LIN {X -0.120,Y -569.299,Z 835.308,A 0.000,B 0.000,C 90.000,E1 91.489} C_DIS
LIN {X -0.052,Y -569.722,Z 835.301,A 0.000,B 0.000,C 90.000,E1 90.115} C_DIS
LIN {X 0.024,Y -570.053,Z 835.293,A 0.000,B 0.000,C 90.000,E1 88.740} C_DIS
LIN {X -0.168,Y -570.463,Z 835.282,A 0.000,B 0.000,C 90.000,E1 86.846} C_DIS
LIN {X 0.104,Y -570.739,Z 835.273,A 0.000,B 0.000,C 90.000,E1 85.179} C_DIS
LIN {X -0.200,Y -571.053,Z 835.264,A 0.000,B 0.000,C 90.000,E1 83.571} C_DIS
LIN {X 0.004,Y -571.342,Z 835.257,A 0.000,B 0.000,C 90.000,E1 82.186} C_DIS
LIN {X -0.074,Y -571.786,Z 835.248,A 0.000,B 0.000,C 90.000,E1 80.557} C_DIS
LIN {X 0.064,Y -572.418,Z 835.237,A 0.000,B 0.000,C 90.000,E1 78.634} C_DIS
LIN {X -0.068,Y -572.823,Z 835.229,A 0.000,B 0.000,C 90.000,E1 77.285} C_DIS
LIN {X -0.005,Y -573.147,Z 835.220,A 0.000,B 0.000,C 90.000,E1 75.644} C_DIS
LIN {X -0.194,Y -573.354,Z 835.214,A 0.000,B 0.000,C 90.000,E1 74.574} C_DIS
LIN {X -0.035,Y -573.431,Z 835.204,A 0.000,B 0.000,C 90.000,E1 72.653} C_DIS
LIN {X 0.133,Y -573.360,Z 835.196,A 0.000,B 0.000,C 90.000,E1 71.275} C_DIS
LIN {X 0.102,Y -573.177,Z 835.187,A 0.000,B 0.000,C 90.000,E1 69.645} C_DIS
LIN {X -0.261,Y -573.034,Z 835.181,A 0.000,B 0.000,C 90.000,E1 68.592} C_DIS
LIN {X -0.090,Y -572.851,Z 835.175,A 0.000,B 0.000,C 90.000,E1 67.486} C_DIS
LIN {X 0.133,Y -572.485,Z 835.167,A 0.000,B 0.000,C 90.000,E1 66.102} C_DIS
LIN {X 0.191,Y -571.841,Z 835.158,A 0.000,B 0.000,C 90.000,E1 64.460} C_DIS
LIN {X -0.118,Y -571.242,Z 835.151,A 0.000,B 0.000,C 90.000,E1 63.127} C_DIS
LIN {X -0.183,Y -570.569,Z 835.143,A 0.000,B 0.000,C 90.000,E1 61.769} C_DIS
LIN {X 0.251,Y -570.332,Z 835.140,A 0.000,B 0.000,C 90.000,E1 61.179} C_DIS
LIN {X -0.159,Y -569.417,Z 835.134,A 0.000,B 0.000,C 90.000,E1 60.127} C_DIS
LIN {X 0.013,Y -568.014,Z 835.126,A 0.000,B 0.000,C 90.000,E1 58.742} C_DIS
LIN {X -0.031,Y -566.388,Z 835.119,A 0.000,B 0.000,C 90.000,E1 57.375} C_DIS
LIN {X -0.208,Y -564.795,Z 835.113,A 0.000,B 0.000,C 90.000,E1 56.294} C_DIS
LIN {X -0.203,Y -563.469,Z 835.108,A 0.000,B 0.000,C 90.000,E1 55.468} C_DIS
LIN {X -0.115,Y -561.414,Z 835.102,A 0.000,B 0.000,C 90.000,E1 54.356} C_DIS
LIN {X 0.176,Y -559.714,Z 835.097,A 0.000,B 0.000,C 90.000,E1 53.497} C_DIS
LIN {X -0.086,Y -558.502,Z 835.094,A 0.000,B 0.000,C 90.000,E1 52.970} C_DIS
LIN {X 0.179,Y -556.410,Z 835.090,A 0.000,B 0.000,C 90.000,E1 52.110} C_DIS
LIN {X -0.019,Y -554.074,Z 835.085,A 0.000,B 0.000,C 90.000,E1 51.295} C_DIS
LIN {X 0.124,Y -552.393,Z 835.082,A 0.000,B 0.000,C 90.000,E1 50.723} C_DIS
LIN {X -0.116,Y -549.571,Z 835.077,A 0.000,B 0.000,C 90.000,E1 49.908} C_DIS
LIN {X -0.027,Y -546.387,Z 835.073,A 0.000,B 0.000,C 90.000,E1 49.057} C_DIS
LIN {X 0.242,Y -543.489,Z 835.069,A 0.000,B 0.000,C 90.000,E1 48.324} C_DIS
LIN {X -0.118,Y -540.968,Z 835.065,A 0.000,B 0.000,C 90.000,E1 47.796} C_DIS
LIN {X -0.130,Y -538.213,Z 835.062,A 0.000,B 0.000,C 90.000,E1 47.229} C_DIS
LIN {X 0.020,Y -534.370,Z 835.058,A 0.000,B 0.000,C 90.000,E1 46.500} C_DIS
LIN {X 0.349,Y -531.058,Z 835.055,A 0.000,B 0.000,C 90.000,E1 45.891} C_DIS
LIN {X 0.268,Y -527.360,Z 835.052,A 0.000,B 0.000,C 90.000,E1 45.324} C_DIS
LIN {X 0.161,Y -523.332,Z 835.049,A 0.000,B 0.000,C 90.000,E1 44.757} C_DIS
LIN {X 0.026,Y -518.943,Z 835.046,A 0.000,B 0.000,C 90.000,E1 44.190} C_DIS
LIN {X -0.024,Y -514.327,Z 835.042,A 0.000,B 0.000,C 90.000,E1 43.623} C_DIS
LIN {X 0.089,Y -510.741,Z 835.040,A 0.000,B 0.000,C 90.000,E1 43.176} C_DIS
LIN {X 0.028,Y -505.522,Z 835.037,A 0.000,B 0.000,C 90.000,E1 42.609} C_DIS
LIN {X -0.024,Y -500.041,Z 835.034,A 0.000,B 0.000,C 90.000,E1 42.043} C_DIS
LIN {X 0.016,Y -496.033,Z 835.031,A 0.000,B 0.000,C 90.000,E1 41.634} C_DIS
LIN {X 0.029,Y -489.092,Z 835.028,A 0.000,B 0.000,C 90.000,E1 40.987} C_DIS
LIN {X 0.092,Y -483.021,Z 835.025,A 0.000,B 0.000,C 90.000,E1 40.458} C_DIS
LIN {X -0.032,Y -475.383,Z 835.021,A 0.000,B 0.000,C 90.000,E1 39.850} C_DIS
LIN {X 0.137,Y -466.165,Z 835.017,A 0.000,B 0.000,C 90.000,E1 39.116} C_DIS
LIN {X 0.072,Y -453.584,Z 835.012,A 0.000,B 0.000,C 90.000,E1 38.177} C_DIS
LIN {X 0.015,Y -440.852,Z 835.007,A 0.000,B 0.000,C 90.000,E1 37.237} C_DIS
LIN {X 0.060,Y -420.752,Z 834.998,A 0.000,B 0.000,C 90.000,E1 35.644} C_DIS
LIN {X 0.124,Y -410.398,Z 834.993,A 0.000,B 0.000,C 90.000,E1 34.739} C_DIS
LIN {X -0.033,Y -404.337,Z 834.990,A 0.000,B 0.000,C 90.000,E1 34.199} C_DIS
LIN {X 0.112,Y -399.570,Z 834.987,A 0.000,B 0.000,C 90.000,E1 33.658} C_DIS
LIN {X 0.091,Y -398.266,Z 834.986,A 0.000,B 0.000,C 90.000,E1 33.499} C_DIS
LIN {X -0.239,Y -395.679,Z 834.984,A 0.000,B 0.000,C 90.000,E1 33.166} C_DIS
LIN {X 0.055,Y -395.661,Z 834.984,A 0.000,B 0.000,C 90.000,E1 33.118} C_DIS
LIN {X 0.091,Y -393.941,Z 834.977,A 0.000,B 0.000,C 90.000,E1 31.926} C_DIS
LIN {X -0.123,Y -391.263,Z 834.970,A 0.000,B 0.000,C 90.000,E1 30.541} C_DIS
LIN {X -0.028,Y -391.514,Z 834.964,A 0.000,B 0.000,C 90.000,E1 29.461} C_DIS
LIN {X -0.208,Y -392.887,Z 834.950,A 0.000,B 0.000,C 90.000,E1 27.001} C_DIS
LIN {X 0.035,Y -394.828,Z 834.934,A 0.000,B 0.000,C 90.000,E1 24.131} C_DIS
LIN {X -0.055,Y -396.510,Z 834.922,A 0.000,B 0.000,C 90.000,E1 22.025} C_DIS
LIN {X -0.016,Y -399.373,Z 834.905,A 0.000,B 0.000,C 90.000,E1 18.852} C_DIS
LIN {X -0.132,Y -402.980,Z 834.887,A 0.000,B 0.000,C 90.000,E1 15.717} C_DIS
LIN {X -0.166,Y -407.456,Z 834.870,A 0.000,B 0.000,C 90.000,E1 12.591} C_DIS
LIN {X 0.029,Y -410.786,Z 834.858,A 0.000,B 0.000,C 90.000,E1 10.489} C_DIS
LIN {X -0.210,Y -413.708,Z 834.849,A 0.000,B 0.000,C 90.000,E1 8.803} C_DIS
LIN {X 0.007,Y -417.352,Z 834.837,A 0.000,B 0.000,C 90.000,E1 6.720} C_DIS
LIN {X -0.070,Y -422.343,Z 834.822,A 0.000,B 0.000,C 90.000,E1 4.012} C_DIS
LIN {X 0.044,Y -429.232,Z 834.804,A 0.000,B 0.000,C 90.000,E1 0.630} C_DIS
LIN {X -0.189,Y -435.722,Z 834.788,A 0.000,B 0.000,C 90.000,E1 357.822} C_DIS
LIN {X 0.132,Y -441.316,Z 834.775,A 0.000,B 0.000,C 90.000,E1 355.469} C_DIS
LIN {X 0.065,Y -446.342,Z 834.764,A 0.000,B 0.000,C 90.000,E1 353.514} C_DIS
LIN {X 0.097,Y -449.017,Z 834.759,A 0.000,B 0.000,C 90.000,E1 352.534} C_DIS
LIN {X -0.037,Y -450.535,Z 834.756,A 0.000,B 0.000,C 90.000,E1 352.064} C_DIS
LIN {X -0.192,Y -453.090,Z 834.753,A 0.000,B 0.000,C 90.000,E1 351.489} C_DIS
LIN {X -0.176,Y -455.431,Z 834.750,A 0.000,B 0.000,C 90.000,E1 351.084} C_DIS
LIN {X -0.065,Y -460.510,Z 834.748,A 0.000,B 0.000,C 90.000,E1 350.557} C_DIS
LIN {X -0.105,Y -466.031,Z 834.745,A 0.000,B 0.000,C 90.000,E1 350.151} C_DIS
LIN {X 0.110,Y -480.162,Z 834.741,A 0.000,B 0.000,C 90.000,E1 349.285} C_DIS
LIN {X 0.120,Y -489.899,Z 834.737,A 0.000,B 0.000,C 90.000,E1 348.701} C_DIS
LIN {X 0.257,Y -496.316,Z 834.735,A 0.000,B 0.000,C 90.000,E1 348.285} C_DIS
LIN {X -0.026,Y -507.454,Z 834.731,A 0.000,B 0.000,C 90.000,E1 347.589} C_DIS
LIN {X 0.093,Y -516.832,Z 834.728,A 0.000,B 0.000,C 90.000,E1 346.937} C_DIS
LIN {X 0.112,Y -527.555,Z 834.723,A 0.000,B 0.000,C 90.000,E1 346.172} C_DIS
LIN {X -0.180,Y -535.027,Z 834.720,A 0.000,B 0.000,C 90.000,E1 345.644} C_DIS
LIN {X 0.184,Y -542.141,Z 834.717,A 0.000,B 0.000,C 90.000,E1 345.046} C_DIS
LIN {X 0.110,Y -549.312,Z 834.714,A 0.000,B 0.000,C 90.000,E1 344.464} C_DIS
LIN {X -0.045,Y -558.907,Z 834.709,A 0.000,B 0.000,C 90.000,E1 343.614} C_DIS
LIN {X -0.022,Y -565.482,Z 834.705,A 0.000,B 0.000,C 90.000,E1 342.960} C_DIS
LIN {X -0.185,Y -571.704,Z 834.702,A 0.000,B 0.000,C 90.000,E1 342.308} C_DIS
LIN {X 0.160,Y -578.789,Z 834.697,A 0.000,B 0.000,C 90.000,E1 341.456} C_DIS
LIN {X 0.191,Y -583.083,Z 834.694,A 0.000,B 0.000,C 90.000,E1 340.913} C_DIS
LIN {X -0.150,Y -590.010,Z 834.689,A 0.000,B 0.000,C 90.000,E1 340.007} C_DIS
LIN {X -0.159,Y -595.400,Z 834.684,A 0.000,B 0.000,C 90.000,E1 339.209} C_DIS
LIN {X -0.110,Y -600.400,Z 834.680,A 0.000,B 0.000,C 90.000,E1 338.411} C_DIS
LIN {X 0.288,Y -603.548,Z 834.677,A 0.000,B 0.000,C 90.000,E1 337.847} C_DIS
LIN {X 0.345,Y -610.264,Z 834.671,A 0.000,B 0.000,C 90.000,E1 336.666} C_DIS
LIN {X -0.032,Y -615.315,Z 834.666,A 0.000,B 0.000,C 90.000,E1 335.793} C_DIS
LIN {X -0.098,Y -620.112,Z 834.661,A 0.000,B 0.000,C 90.000,E1 334.897} C_DIS
LIN {X 0.184,Y -623.975,Z 834.656,A 0.000,B 0.000,C 90.000,E1 334.101} C_DIS
LIN {X 0.211,Y -627.690,Z 834.652,A 0.000,B 0.000,C 90.000,E1 333.332} C_DIS
LIN {X -0.262,Y -632.292,Z 834.646,A 0.000,B 0.000,C 90.000,E1 332.359} C_DIS
LIN {X 0.230,Y -637.757,Z 834.639,A 0.000,B 0.000,C 90.000,E1 331.051} C_DIS
LIN {X -0.174,Y -640.869,Z 834.635,A 0.000,B 0.000,C 90.000,E1 330.333} C_DIS
LIN {X -0.096,Y -645.795,Z 834.628,A 0.000,B 0.000,C 90.000,E1 329.076} C_DIS
LIN {X -0.020,Y -649.321,Z 834.623,A 0.000,B 0.000,C 90.000,E1 328.074} C_DIS
LIN {X -0.014,Y -653.497,Z 834.616,A 0.000,B 0.000,C 90.000,E1 326.834} C_DIS
LIN {X 0.062,Y -655.742,Z 834.612,A 0.000,B 0.000,C 90.000,E1 326.087} C_DIS
LIN {X 0.083,Y -658.634,Z 834.606,A 0.000,B 0.000,C 90.000,E1 325.102} C_DIS
LIN {X 0.145,Y -661.300,Z 834.601,A 0.000,B 0.000,C 90.000,E1 324.116} C_DIS
LIN {X -0.251,Y -663.053,Z 834.597,A 0.000,B 0.000,C 90.000,E1 323.417} C_DIS
LIN {X 0.263,Y -665.237,Z 834.591,A 0.000,B 0.000,C 90.000,E1 322.396} C_DIS
LIN {X -0.125,Y -667.211,Z 834.586,A 0.000,B 0.000,C 90.000,E1 321.457} C_DIS
LIN {X -0.069,Y -668.989,Z 834.580,A 0.000,B 0.000,C 90.000,E1 320.481} C_DIS
LIN {X 0.090,Y -670.998,Z 834.574,A 0.000,B 0.000,C 90.000,E1 319.256} C_DIS
LIN {X 0.230,Y -673.653,Z 834.564,A 0.000,B 0.000,C 90.000,E1 317.553} C_DIS
LIN {X -0.165,Y -674.737,Z 834.560,A 0.000,B 0.000,C 90.000,E1 316.863} C_DIS
LIN {X 0.035,Y -676.870,Z 834.551,A 0.000,B 0.000,C 90.000,E1 315.162} C_DIS
LIN {X 0.212,Y -678.249,Z 834.544,A 0.000,B 0.000,C 90.000,E1 313.947} C_DIS
LIN {X -0.020,Y -679.817,Z 834.536,A 0.000,B 0.000,C 90.000,E1 312.528} C_DIS
LIN {X 0.279,Y -681.355,Z 834.528,A 0.000,B 0.000,C 90.000,E1 311.067} C_DIS
LIN {X 0.119,Y -682.528,Z 834.522,A 0.000,B 0.000,C 90.000,E1 309.886} C_DIS
LIN {X -0.014,Y -683.593,Z 834.515,A 0.000,B 0.000,C 90.000,E1 308.705} C_DIS
LIN {X -0.135,Y -684.639,Z 834.508,A 0.000,B 0.000,C 90.000,E1 307.523} C_DIS
LIN {X 0.297,Y -685.662,Z 834.502,A 0.000,B 0.000,C 90.000,E1 306.297} C_DIS
LIN {X 0.340,Y -686.618,Z 834.495,A 0.000,B 0.000,C 90.000,E1 305.105} C_DIS
LIN {X 0.027,Y -687.625,Z 834.487,A 0.000,B 0.000,C 90.000,E1 303.706} C_DIS
LIN {X -0.073,Y -688.603,Z 834.479,A 0.000,B 0.000,C 90.000,E1 302.291} C_DIS
LIN {X 0.433,Y -689.807,Z 834.470,A 0.000,B 0.000,C 90.000,E1 300.590} C_DIS
LIN {X 0.021,Y -690.884,Z 834.462,A 0.000,B 0.000,C 90.000,E1 299.205} C_DIS
LIN {X -0.006,Y -691.825,Z 834.456,A 0.000,B 0.000,C 90.000,E1 298.025} C_DIS
LIN {X -0.227,Y -693.391,Z 834.445,A 0.000,B 0.000,C 90.000,E1 296.155} C_DIS
LIN {X 0.292,Y -694.802,Z 834.436,A 0.000,B 0.000,C 90.000,E1 294.463} C_DIS
LIN {X 0.126,Y -695.027,Z 834.432,A 0.000,B 0.000,C 90.000,E1 293.770} C_DIS
LIN {X -0.290,Y -694.417,Z 834.430,A 0.000,B 0.000,C 90.000,E1 293.334} C_DIS
LIN {X -0.042,Y -693.967,Z 834.428,A 0.000,B 0.000,C 90.000,E1 293.078} C_DIS
LIN {X 0.056,Y -692.154,Z 834.426,A 0.000,B 0.000,C 90.000,E1 292.717} C_DIS
LIN {X 0.295,Y -690.711,Z 834.425,A 0.000,B 0.000,C 90.000,E1 292.461} C_DIS
LIN {X -0.226,Y -689.876,Z 834.424,A 0.000,B 0.000,C 90.000,E1 292.386} C_DIS
LIN {X -0.111,Y -688.662,Z 834.424,A 0.000,B 0.000,C 90.000,E1 292.259} C_DIS
LIN {X -0.186,Y -684.038,Z 834.422,A 0.000,B 0.000,C 90.000,E1 291.950} C_DIS
LIN {X -0.073,Y -682.425,Z 834.421,A 0.000,B 0.000,C 90.000,E1 291.844} C_DIS
LIN {X 0.292,Y -680.489,Z 834.421,A 0.000,B 0.000,C 90.000,E1 291.716} C_DIS
LIN {X 0.211,Y -671.837,Z 834.419,A 0.000,B 0.000,C 90.000,E1 291.461} C_DIS
LIN {X 0.243,Y -663.448,Z 834.418,A 0.000,B 0.000,C 90.000,E1 291.280} C_DIS
LIN {X 0.212,Y -655.251,Z 834.418,A 0.000,B 0.000,C 90.000,E1 291.153} C_DIS
LIN {X 0.175,Y -646.300,Z 834.417,A 0.000,B 0.000,C 90.000,E1 290.972} C_DIS
LIN {X 0.364,Y -639.749,Z 834.416,A 0.000,B 0.000,C 90.000,E1 290.791} C_DIS
LIN {X 0.255,Y -635.161,Z 834.415,A 0.000,B 0.000,C 90.000,E1 290.663} C_DIS
LIN {X -0.113,Y -631.474,Z 834.414,A 0.000,B 0.000,C 90.000,E1 290.556} C_DIS
LIN {X -0.036,Y -626.194,Z 834.413,A 0.000,B 0.000,C 90.000,E1 290.301} C_DIS
LIN {X -0.165,Y -625.101,Z 834.412,A 0.000,B 0.000,C 90.000,E1 290.248} C_DIS
LIN {X 0.250,Y -623.492,Z 834.412,A 0.000,B 0.000,C 90.000,E1 290.066} C_DIS
LIN {X 0.217,Y -623.471,Z 834.412,A 0.000,B 0.000,C 90.000,E1 290.066} C_DIS
LIN {X 0.049,Y -623.220,Z 834.411,A 0.000,B 0.000,C 90.000,E1 289.939} C_DIS
LIN {X -0.061,Y -623.280,Z 834.411,A 0.000,B 0.000,C 90.000,E1 289.885} C_DIS
LIN {X -0.190,Y -624.798,Z 834.408,A 0.000,B 0.000,C 90.000,E1 289.450} C_DIS
LIN {X -0.067,Y -629.481,Z 834.403,A 0.000,B 0.000,C 90.000,E1 288.598} C_DIS
LIN {X -0.155,Y -632.392,Z 834.401,A 0.000,B 0.000,C 90.000,E1 288.109} C_DIS
LIN {X 0.128,Y -636.087,Z 834.396,A 0.000,B 0.000,C 90.000,E1 287.330} C_DIS
LIN {X -0.232,Y -638.364,Z 834.394,A 0.000,B 0.000,C 90.000,E1 286.858} C_DIS
LIN {X 0.055,Y -641.172,Z 834.389,A 0.000,B 0.000,C 90.000,E1 286.079} C_DIS
LIN {X 0.197,Y -643.583,Z 834.385,A 0.000,B 0.000,C 90.000,E1 285.315} C_DIS
LIN {X 0.061,Y -644.904,Z 834.382,A 0.000,B 0.000,C 90.000,E1 284.828} C_DIS
LIN {X 0.246,Y -646.463,Z 834.378,A 0.000,B 0.000,C 90.000,E1 284.064} C_DIS
LIN {X -0.039,Y -647.380,Z 834.376,A 0.000,B 0.000,C 90.000,E1 283.592} C_DIS
LIN {X 0.313,Y -647.948,Z 834.373,A 0.000,B 0.000,C 90.000,E1 283.063} C_DIS
LIN {X -0.100,Y -648.147,Z 834.369,A 0.000,B 0.000,C 90.000,E1 282.355} C_DIS
LIN {X 0.256,Y -648.026,Z 834.366,A 0.000,B 0.000,C 90.000,E1 281.827} C_DIS
LIN {X -0.151,Y -647.731,Z 834.363,A 0.000,B 0.000,C 90.000,E1 281.366} C_DIS
LIN {X 0.061,Y -646.822,Z 834.359,A 0.000,B 0.000,C 90.000,E1 280.602} C_DIS
LIN {X -0.344,Y -645.875,Z 834.356,A 0.000,B 0.000,C 90.000,E1 280.141} C_DIS
LIN {X -0.005,Y -644.634,Z 834.353,A 0.000,B 0.000,C 90.000,E1 279.613} C_DIS
LIN {X 0.217,Y -642.910,Z 834.351,A 0.000,B 0.000,C 90.000,E1 279.095} C_DIS
LIN {X -0.107,Y -640.802,Z 834.348,A 0.000,B 0.000,C 90.000,E1 278.624} C_DIS
LIN {X 0.094,Y -638.380,Z 834.345,A 0.000,B 0.000,C 90.000,E1 278.106} C_DIS
LIN {X -0.221,Y -636.307,Z 834.343,A 0.000,B 0.000,C 90.000,E1 277.757} C_DIS
LIN {X 0.085,Y -633.884,Z 834.341,A 0.000,B 0.000,C 90.000,E1 277.352} C_DIS
LIN {X 0.093,Y -629.125,Z 834.337,A 0.000,B 0.000,C 90.000,E1 276.720} C_DIS
LIN {X -0.263,Y -625.775,Z 834.335,A 0.000,B 0.000,C 90.000,E1 276.372} C_DIS
LIN {X 0.212,Y -624.546,Z 834.335,A 0.000,B 0.000,C 90.000,E1 276.201} C_DIS
LIN {X 0.028,Y -619.077,Z 834.332,A 0.000,B 0.000,C 90.000,E1 275.739} C_DIS
LIN {X 0.263,Y -613.057,Z 834.330,A 0.000,B 0.000,C 90.000,E1 275.277} C_DIS
LIN {X -0.060,Y -609.758,Z 834.328,A 0.000,B 0.000,C 90.000,E1 275.106} C_DIS
LIN {X 0.103,Y -604.710,Z 834.327,A 0.000,B 0.000,C 90.000,E1 274.821} C_DIS
LIN {X -0.280,Y -597.826,Z 834.325,A 0.000,B 0.000,C 90.000,E1 274.531} C_DIS
LIN {X 0.231,Y -590.869,Z 834.323,A 0.000,B 0.000,C 90.000,E1 274.188} C_DIS
LIN {X -0.065,Y -585.648,Z 834.322,A 0.000,B 0.000,C 90.000,E1 274.012} C_DIS
LIN {X -0.120,Y -579.728,Z 834.321,A 0.000,B 0.000,C 90.000,E1 273.841} C_DIS
LIN {X -0.062,Y -577.758,Z 834.321,A 0.000,B 0.000,C 90.000,E1 273.784} C_DIS
LIN {X -0.149,Y -571.161,Z 834.320,A 0.000,B 0.000,C 90.000,E1 273.669} C_DIS
LIN {X -0.186,Y -564.612,Z 834.320,A 0.000,B 0.000,C 90.000,E1 273.612} C_DIS
LIN {X 0.085,Y -553.744,Z 834.320,A 0.000,B 0.000,C 90.000,E1 273.555} C_DIS
LIN {X -0.236,Y -552.354,Z 834.320,A 0.000,B 0.000,C 90.000,E1 273.555} C_DIS
LIN {X 0.260,Y -550.562,Z 834.319,A 0.000,B 0.000,C 90.000,E1 273.440} C_DIS
LIN {X 0.217,Y -550.542,Z 834.319,A 0.000,B 0.000,C 90.000,E1 273.440} C_DIS
LIN {X -0.216,Y -549.459,Z 834.318,A 0.000,B 0.000,C 90.000,E1 273.212} C_DIS
LIN {X 0.099,Y -548.692,Z 834.316,A 0.000,B 0.000,C 90.000,E1 272.808} C_DIS
LIN {X -0.191,Y -547.087,Z 834.308,A 0.000,B 0.000,C 90.000,E1 271.432} C_DIS
LIN {X 0.191,Y -545.161,Z 834.294,A 0.000,B 0.000,C 90.000,E1 268.854} C_DIS
LIN {X -0.123,Y -543.975,Z 834.284,A 0.000,B 0.000,C 90.000,E1 267.192} C_DIS
LIN {X 0.086,Y -543.031,Z 834.276,A 0.000,B 0.000,C 90.000,E1 265.755} C_DIS
LIN {X -0.245,Y -541.924,Z 834.267,A 0.000,B 0.000,C 90.000,E1 264.090} C_DIS
LIN {X -0.097,Y -541.269,Z 834.262,A 0.000,B 0.000,C 90.000,E1 263.223} C_DIS
LIN {X 0.113,Y -539.960,Z 834.254,A 0.000,B 0.000,C 90.000,E1 261.781} C_DIS
LIN {X -0.089,Y -538.416,Z 834.245,A 0.000,B 0.000,C 90.000,E1 260.095} C_DIS
LIN {X 0.306,Y -536.679,Z 834.235,A 0.000,B 0.000,C 90.000,E1 258.342} C_DIS
LIN {X 0.135,Y -534.959,Z 834.226,A 0.000,B 0.000,C 90.000,E1 256.645} C_DIS
LIN {X -0.051,Y -533.642,Z 834.220,A 0.000,B 0.000,C 90.000,E1 255.519} C_DIS
LIN {X -0.216,Y -532.003,Z 834.212,A 0.000,B 0.000,C 90.000,E1 254.102} C_DIS
LIN {X -0.115,Y -530.321,Z 834.204,A 0.000,B 0.000,C 90.000,E1 252.653} C_DIS
LIN {X 0.287,Y -528.962,Z 834.197,A 0.000,B 0.000,C 90.000,E1 251.456} C_DIS
LIN {X 0.157,Y -527.447,Z 834.191,A 0.000,B 0.000,C 90.000,E1 250.315} C_DIS
LIN {X -0.144,Y -525.445,Z 834.183,A 0.000,B 0.000,C 90.000,E1 248.901} C_DIS
LIN {X 0.051,Y -522.569,Z 834.171,A 0.000,B 0.000,C 90.000,E1 246.847} C_DIS
LIN {X -0.127,Y -520.299,Z 834.163,A 0.000,B 0.000,C 90.000,E1 245.409} C_DIS
LIN {X -0.026,Y -518.493,Z 834.157,A 0.000,B 0.000,C 90.000,E1 244.229} C_DIS
LIN {X 0.033,Y -516.490,Z 834.150,A 0.000,B 0.000,C 90.000,E1 243.050} C_DIS
LIN {X -0.154,Y -513.368,Z 834.141,A 0.000,B 0.000,C 90.000,E1 241.307} C_DIS
LIN {X 0.187,Y -510.651,Z 834.132,A 0.000,B 0.000,C 90.000,E1 239.793} C_DIS
LIN {X 0.135,Y -508.458,Z 834.126,A 0.000,B 0.000,C 90.000,E1 238.614} C_DIS
LIN {X -0.119,Y -506.168,Z 834.119,A 0.000,B 0.000,C 90.000,E1 237.454} C_DIS
LIN {X -0.096,Y -503.039,Z 834.111,A 0.000,B 0.000,C 90.000,E1 235.960} C_DIS
LIN {X -0.147,Y -500.340,Z 834.104,A 0.000,B 0.000,C 90.000,E1 234.769} C_DIS
LIN {X 0.194,Y -496.097,Z 834.094,A 0.000,B 0.000,C 90.000,E1 232.924} C_DIS
LIN {X -0.055,Y -493.286,Z 834.087,A 0.000,B 0.000,C 90.000,E1 231.743} C_DIS
LIN {X 0.026,Y -487.613,Z 834.074,A 0.000,B 0.000,C 90.000,E1 229.299} C_DIS
LIN {X -0.026,Y -484.748,Z 834.067,A 0.000,B 0.000,C 90.000,E1 228.081} C_DIS
LIN {X 0.261,Y -479.909,Z 834.055,A 0.000,B 0.000,C 90.000,E1 225.891} C_DIS
LIN {X 0.295,Y -475.883,Z 834.045,A 0.000,B 0.000,C 90.000,E1 224.028} C_DIS
LIN {X 0.115,Y -470.519,Z 834.031,A 0.000,B 0.000,C 90.000,E1 221.553} C_DIS
LIN {X -0.056,Y -466.560,Z 834.021,A 0.000,B 0.000,C 90.000,E1 219.688} C_DIS
LIN {X 0.201,Y -461.956,Z 834.008,A 0.000,B 0.000,C 90.000,E1 217.443} C_DIS
LIN {X -0.167,Y -459.350,Z 834.001,A 0.000,B 0.000,C 90.000,E1 216.217} C_DIS
LIN {X 0.005,Y -455.293,Z 833.990,A 0.000,B 0.000,C 90.000,E1 214.278} C_DIS
LIN {X 0.082,Y -451.104,Z 833.980,A 0.000,B 0.000,C 90.000,E1 212.339} C_DIS
LIN {X -0.042,Y -449.157,Z 833.974,A 0.000,B 0.000,C 90.000,E1 211.386} C_DIS
LIN {X 0.087,Y -443.815,Z 833.960,A 0.000,B 0.000,C 90.000,E1 208.771} C_DIS
LIN {X 0.137,Y -440.538,Z 833.951,A 0.000,B 0.000,C 90.000,E1 207.129} C_DIS
LIN {X 0.049,Y -438.620,Z 833.945,A 0.000,B 0.000,C 90.000,E1 206.155} C_DIS
LIN {X -0.014,Y -435.294,Z 833.936,A 0.000,B 0.000,C 90.000,E1 204.515} C_DIS
LIN {X -0.111,Y -430.601,Z 833.923,A 0.000,B 0.000,C 90.000,E1 202.206} C_DIS
LIN {X -0.107,Y -427.413,Z 833.914,A 0.000,B 0.000,C 90.000,E1 200.536} C_DIS
LIN {X -0.059,Y -424.108,Z 833.905,A 0.000,B 0.000,C 90.000,E1 198.852} C_DIS
LIN {X -0.117,Y -419.551,Z 833.892,A 0.000,B 0.000,C 90.000,E1 196.496} C_DIS
LIN {X 0.063,Y -416.341,Z 833.882,A 0.000,B 0.000,C 90.000,E1 194.773} C_DIS
LIN {X 0.035,Y -413.644,Z 833.875,A 0.000,B 0.000,C 90.000,E1 193.411} C_DIS
LIN {X 0.037,Y -408.947,Z 833.861,A 0.000,B 0.000,C 90.000,E1 191.007} C_DIS
LIN {X 0.146,Y -405.024,Z 833.850,A 0.000,B 0.000,C 90.000,E1 188.916} C_DIS
LIN {X 0.107,Y -401.727,Z 833.840,A 0.000,B 0.000,C 90.000,E1 187.182} C_DIS
LIN {X -0.063,Y -397.811,Z 833.828,A 0.000,B 0.000,C 90.000,E1 185.106} C_DIS
LIN {X -0.182,Y -392.728,Z 833.811,A 0.000,B 0.000,C 90.000,E1 181.949} C_DIS
LIN {X -0.118,Y -388.474,Z 833.793,A 0.000,B 0.000,C 90.000,E1 178.740} C_DIS
LIN {X 0.113,Y -385.774,Z 833.781,A 0.000,B 0.000,C 90.000,E1 176.560} C_DIS
LIN {X 0.006,Y -383.520,Z 833.771,A 0.000,B 0.000,C 90.000,E1 174.780} C_DIS
LIN {X -0.099,Y -379.716,Z 833.753,A 0.000,B 0.000,C 90.000,E1 171.546} C_DIS
LIN {X 0.076,Y -377.590,Z 833.741,A 0.000,B 0.000,C 90.000,E1 169.342} C_DIS
LIN {X 0.103,Y -376.216,Z 833.733,A 0.000,B 0.000,C 90.000,E1 167.881} C_DIS
LIN {X 0.043,Y -374.423,Z 833.721,A 0.000,B 0.000,C 90.000,E1 165.700} C_DIS
LIN {X -0.083,Y -372.392,Z 833.700,A 0.000,B 0.000,C 90.000,E1 162.054} C_DIS
LIN {X 0.112,Y -372.343,Z 833.690,A 0.000,B 0.000,C 90.000,E1 160.188} C_DIS
LIN {X 0.074,Y -372.979,Z 833.680,A 0.000,B 0.000,C 90.000,E1 158.358} C_DIS
LIN {X -0.127,Y -374.178,Z 833.672,A 0.000,B 0.000,C 90.000,E1 156.922} C_DIS
LIN {X -0.047,Y -375.131,Z 833.668,A 0.000,B 0.000,C 90.000,E1 156.177} C_DIS
LIN {X 0.039,Y -376.442,Z 833.664,A 0.000,B 0.000,C 90.000,E1 155.433} C_DIS
LIN {X -0.040,Y -378.226,Z 833.660,A 0.000,B 0.000,C 90.000,E1 154.717} C_DIS
LIN {X 0.094,Y -379.258,Z 833.658,A 0.000,B 0.000,C 90.000,E1 154.332} C_DIS
LIN {X -0.113,Y -381.666,Z 833.654,A 0.000,B 0.000,C 90.000,E1 153.640} C_DIS
LIN {X 0.167,Y -383.622,Z 833.651,A 0.000,B 0.000,C 90.000,E1 153.127} C_DIS
LIN {X -0.016,Y -385.534,Z 833.649,A 0.000,B 0.000,C 90.000,E1 152.794} C_DIS
LIN {X 0.147,Y -389.402,Z 833.646,A 0.000,B 0.000,C 90.000,E1 152.231} C_DIS
LIN {X -0.010,Y -392.176,Z 833.644,A 0.000,B 0.000,C 90.000,E1 151.897} C_DIS
LIN {X 0.171,Y -397.794,Z 833.641,A 0.000,B 0.000,C 90.000,E1 151.385} C_DIS
LIN {X -0.078,Y -399.358,Z 833.641,A 0.000,B 0.000,C 90.000,E1 151.307} C_DIS
LIN {X 0.004,Y -407.973,Z 833.638,A 0.000,B 0.000,C 90.000,E1 150.845} C_DIS
LIN {X -0.197,Y -414.984,Z 833.637,A 0.000,B 0.000,C 90.000,E1 150.589} C_DIS
LIN {X 0.025,Y -421.820,Z 833.635,A 0.000,B 0.000,C 90.000,E1 150.255} C_DIS
LIN {X 0.069,Y -428.530,Z 833.633,A 0.000,B 0.000,C 90.000,E1 149.921} C_DIS
LIN {X -0.106,Y -434.975,Z 833.631,A 0.000,B 0.000,C 90.000,E1 149.587} C_DIS
LIN {X -0.156,Y -442.701,Z 833.628,A 0.000,B 0.000,C 90.000,E1 149.076} C_DIS
LIN {X 0.128,Y -450.368,Z 833.625,A 0.000,B 0.000,C 90.000,E1 148.456} C_DIS
LIN {X -0.150,Y -456.446,Z 833.622,A 0.000,B 0.000,C 90.000,E1 147.995} C_DIS
LIN {X 0.045,Y -459.633,Z 833.621,A 0.000,B 0.000,C 90.000,E1 147.709} C_DIS
LIN {X 0.083,Y -466.471,Z 833.617,A 0.000,B 0.000,C 90.000,E1 147.041} C_DIS
LIN {X -0.207,Y -474.829,Z 833.612,A 0.000,B 0.000,C 90.000,E1 146.215} C_DIS
LIN {X 0.063,Y -480.226,Z 833.609,A 0.000,B 0.000,C 90.000,E1 145.595} C_DIS
LIN {X -0.257,Y -484.123,Z 833.606,A 0.000,B 0.000,C 90.000,E1 145.182} C_DIS
LIN {X 0.191,Y -493.061,Z 833.600,A 0.000,B 0.000,C 90.000,E1 143.909} C_DIS
LIN {X -0.103,Y -497.392,Z 833.596,A 0.000,B 0.000,C 90.000,E1 143.336} C_DIS
LIN {X 0.030,Y -501.413,Z 833.593,A 0.000,B 0.000,C 90.000,E1 142.718} C_DIS
LIN {X 0.099,Y -505.326,Z 833.590,A 0.000,B 0.000,C 90.000,E1 142.110} C_DIS
LIN {X -0.009,Y -507.425,Z 833.588,A 0.000,B 0.000,C 90.000,E1 141.823} C_DIS
LIN {X -0.092,Y -511.921,Z 833.584,A 0.000,B 0.000,C 90.000,E1 141.090} C_DIS
LIN {X 0.057,Y -519.721,Z 833.576,A 0.000,B 0.000,C 90.000,E1 139.747} C_DIS
LIN {X 0.137,Y -522.156,Z 833.574,A 0.000,B 0.000,C 90.000,E1 139.299} C_DIS
LIN {X 0.034,Y -525.230,Z 833.571,A 0.000,B 0.000,C 90.000,E1 138.728} C_DIS
LIN {X -0.256,Y -527.743,Z 833.568,A 0.000,B 0.000,C 90.000,E1 138.324} C_DIS
LIN {X -0.061,Y -533.668,Z 833.562,A 0.000,B 0.000,C 90.000,E1 137.148} C_DIS
LIN {X 0.018,Y -544.722,Z 833.550,A 0.000,B 0.000,C 90.000,E1 135.000} C_DIS
LIN {X -0.333,Y -549.096,Z 833.545,A 0.000,B 0.000,C 90.000,E1 134.190} C_DIS
LIN {X 0.135,Y -553.102,Z 833.541,A 0.000,B 0.000,C 90.000,E1 133.299} C_DIS
LIN {X -0.002,Y -559.474,Z 833.533,A 0.000,B 0.000,C 90.000,E1 131.919} C_DIS
LIN {X -0.031,Y -562.422,Z 833.529,A 0.000,B 0.000,C 90.000,E1 131.229} C_DIS
LIN {X 0.306,Y -567.068,Z 833.523,A 0.000,B 0.000,C 90.000,E1 130.092} C_DIS
LIN {X 0.220,Y -570.376,Z 833.518,A 0.000,B 0.000,C 90.000,E1 129.277} C_DIS
LIN {X 0.033,Y -572.318,Z 833.515,A 0.000,B 0.000,C 90.000,E1 128.749} C_DIS
LIN {X 0.141,Y -576.120,Z 833.509,A 0.000,B 0.000,C 90.000,E1 127.649} C_DIS
LIN {X 0.096,Y -577.808,Z 833.506,A 0.000,B 0.000,C 90.000,E1 127.111} C_DIS
LIN {X 0.279,Y -580.596,Z 833.500,A 0.000,B 0.000,C 90.000,E1 126.011} C_DIS
LIN {X -0.023,Y -582.355,Z 833.496,A 0.000,B 0.000,C 90.000,E1 125.231} C_DIS
LIN {X 0.347,Y -584.427,Z 833.490,A 0.000,B 0.000,C 90.000,E1 124.119} C_DIS
LIN {X -0.106,Y -585.219,Z 833.487,A 0.000,B 0.000,C 90.000,E1 123.627} C_DIS
LIN {X -0.150,Y -586.982,Z 833.479,A 0.000,B 0.000,C 90.000,E1 122.291} C_DIS
LIN {X -0.092,Y -587.545,Z 833.476,A 0.000,B 0.000,C 90.000,E1 121.750} C_DIS
LIN {X 0.031,Y -587.998,Z 833.470,A 0.000,B 0.000,C 90.000,E1 120.669} C_DIS
LIN {X -0.023,Y -588.136,Z 833.466,A 0.000,B 0.000,C 90.000,E1 119.873} C_DIS
LIN {X -0.078,Y -588.071,Z 833.462,A 0.000,B 0.000,C 90.000,E1 119.077} C_DIS
LIN {X -0.139,Y -587.696,Z 833.457,A 0.000,B 0.000,C 90.000,E1 118.281} C_DIS
LIN {X 0.152,Y -587.250,Z 833.454,A 0.000,B 0.000,C 90.000,E1 117.719} C_DIS
LIN {X 0.076,Y -586.190,Z 833.450,A 0.000,B 0.000,C 90.000,E1 116.924} C_DIS
LIN {X -0.160,Y -585.863,Z 833.447,A 0.000,B 0.000,C 90.000,E1 116.411} C_DIS
LIN {X 0.127,Y -585.132,Z 833.444,A 0.000,B 0.000,C 90.000,E1 115.848} C_DIS
LIN {X 0.033,Y -582.433,Z 833.436,A 0.000,B 0.000,C 90.000,E1 114.515} C_DIS
LIN {X 0.299,Y -580.630,Z 833.433,A 0.000,B 0.000,C 90.000,E1 113.951} C_DIS
LIN {X 0.162,Y -579.379,Z 833.432,A 0.000,B 0.000,C 90.000,E1 113.695} C_DIS
LIN {X -0.282,Y -577.191,Z 833.430,A 0.000,B 0.000,C 90.000,E1 113.334} C_DIS
LIN {X 0.024,Y -574.653,Z 833.427,A 0.000,B 0.000,C 90.000,E1 112.898} C_DIS
LIN {X -0.134,Y -572.614,Z 833.426,A 0.000,B 0.000,C 90.000,E1 112.642} C_DIS
LIN {X 0.264,Y -569.471,Z 833.424,A 0.000,B 0.000,C 90.000,E1 112.206} C_DIS
LIN {X -0.041,Y -565.827,Z 833.421,A 0.000,B 0.000,C 90.000,E1 111.844} C_DIS
LIN {X -0.258,Y -564.660,Z 833.420,A 0.000,B 0.000,C 90.000,E1 111.589} C_DIS
LIN {X 0.170,Y -564.031,Z 833.419,A 0.000,B 0.000,C 90.000,E1 111.408} C_DIS
LIN {X 0.161,Y -563.388,Z 833.416,A 0.000,B 0.000,C 90.000,E1 110.791} C_DIS
LIN {X -0.127,Y -563.039,Z 833.411,A 0.000,B 0.000,C 90.000,E1 109.993} C_DIS
LIN {X -0.062,Y -562.071,Z 833.400,A 0.000,B 0.000,C 90.000,E1 108.055} C_DIS
LIN {X 0.009,Y -562.271,Z 833.383,A 0.000,B 0.000,C 90.000,E1 105.009} C_DIS
LIN {X -0.091,Y -563.396,Z 833.370,A 0.000,B 0.000,C 90.000,E1 102.535} C_DIS
LIN {X -0.055,Y -564.646,Z 833.359,A 0.000,B 0.000,C 90.000,E1 100.602} C_DIS
LIN {X 0.124,Y -565.677,Z 833.351,A 0.000,B 0.000,C 90.000,E1 99.208} C_DIS
LIN {X -0.153,Y -566.791,Z 833.342,A 0.000,B 0.000,C 90.000,E1 97.587} C_DIS
LIN {X 0.148,Y -567.754,Z 833.333,A 0.000,B 0.000,C 90.000,E1 95.910} C_DIS
LIN {X 0.237,Y -568.423,Z 833.325,A 0.000,B 0.000,C 90.000,E1 94.531} C_DIS
LIN {X -0.265,Y -568.984,Z 833.318,A 0.000,B 0.000,C 90.000,E1 93.212} C_DIS
LIN {X 0.089,Y -569.608,Z 833.307,A 0.000,B 0.000,C 90.000,E1 91.260} C_DIS
LIN {X 0.163,Y -569.992,Z 833.299,A 0.000,B 0.000,C 90.000,E1 89.885} C_DIS
LIN {X 0.243,Y -570.337,Z 833.292,A 0.000,B 0.000,C 90.000,E1 88.511} C_DIS
LIN {X -0.102,Y -570.673,Z 833.283,A 0.000,B 0.000,C 90.000,E1 86.906} C_DIS
LIN {X 0.159,Y -570.972,Z 833.274,A 0.000,B 0.000,C 90.000,E1 85.241} C_DIS
LIN {X 0.090,Y -571.347,Z 833.263,A 0.000,B 0.000,C 90.000,E1 83.337} C_DIS
LIN {X -0.259,Y -571.627,Z 833.255,A 0.000,B 0.000,C 90.000,E1 82.008} C_DIS
LIN {X -0.225,Y -572.163,Z 833.245,A 0.000,B 0.000,C 90.000,E1 80.095} C_DIS
LIN {X -0.283,Y -572.723,Z 833.236,A 0.000,B 0.000,C 90.000,E1 78.465} C_DIS
LIN {X -0.057,Y -572.995,Z 833.230,A 0.000,B 0.000,C 90.000,E1 77.353} C_DIS
LIN {X 0.140,Y -573.339,Z 833.221,A 0.000,B 0.000,C 90.000,E1 75.700} C_DIS
LIN {X -0.043,Y -573.536,Z 833.215,A 0.000,B 0.000,C 90.000,E1 74.629} C_DIS
LIN {X -0.046,Y -573.589,Z 833.204,A 0.000,B 0.000,C 90.000,E1 72.725} C_DIS
LIN {X -0.066,Y -573.473,Z 833.195,A 0.000,B 0.000,C 90.000,E1 71.094} C_DIS
LIN {X -0.272,Y -573.245,Z 833.184,A 0.000,B 0.000,C 90.000,E1 69.209} C_DIS
LIN {X -0.097,Y -573.030,Z 833.178,A 0.000,B 0.000,C 90.000,E1 68.103} C_DIS
LIN {X 0.070,Y -572.772,Z 833.172,A 0.000,B 0.000,C 90.000,E1 66.997} C_DIS
LIN {X -0.069,Y -572.460,Z 833.166,A 0.000,B 0.000,C 90.000,E1 65.921} C_DIS
LIN {X 0.148,Y -571.950,Z 833.159,A 0.000,B 0.000,C 90.000,E1 64.537} C_DIS
LIN {X 0.092,Y -571.352,Z 833.151,A 0.000,B 0.000,C 90.000,E1 63.179} C_DIS
LIN {X 0.035,Y -570.645,Z 833.143,A 0.000,B 0.000,C 90.000,E1 61.820} C_DIS
LIN {X 0.026,Y -570.159,Z 833.139,A 0.000,B 0.000,C 90.000,E1 61.001} C_DIS
LIN {X -0.216,Y -569.432,Z 833.134,A 0.000,B 0.000,C 90.000,E1 60.205} C_DIS
LIN {X 0.135,Y -568.306,Z 833.128,A 0.000,B 0.000,C 90.000,E1 59.076} C_DIS
LIN {X 0.096,Y -566.701,Z 833.121,A 0.000,B 0.000,C 90.000,E1 57.709} C_DIS
LIN {X -0.183,Y -565.590,Z 833.116,A 0.000,B 0.000,C 90.000,E1 56.914} C_DIS
LIN {X -0.062,Y -563.908,Z 833.110,A 0.000,B 0.000,C 90.000,E1 55.801} C_DIS
LIN {X 0.036,Y -561.922,Z 833.104,A 0.000,B 0.000,C 90.000,E1 54.689} C_DIS
LIN {X 0.099,Y -559.626,Z 833.098,A 0.000,B 0.000,C 90.000,E1 53.577} C_DIS
LIN {X -0.164,Y -558.410,Z 833.095,A 0.000,B 0.000,C 90.000,E1 53.050} C_DIS
LIN {X 0.098,Y -556.294,Z 833.090,A 0.000,B 0.000,C 90.000,E1 52.190} C_DIS
LIN {X -0.102,Y -553.932,Z 833.085,A 0.000,B 0.000,C 90.000,E1 51.376} C_DIS
LIN {X 0.104,Y -551.288,Z 833.081,A 0.000,B 0.000,C 90.000,E1 50.517} C_DIS
LIN {X -0.203,Y -549.401,Z 833.078,A 0.000,B 0.000,C 90.000,E1 49.989} C_DIS
LIN {X -0.117,Y -546.176,Z 833.073,A 0.000,B 0.000,C 90.000,E1 49.138} C_DIS
LIN {X 0.150,Y -543.275,Z 833.069,A 0.000,B 0.000,C 90.000,E1 48.405} C_DIS
LIN {X 0.151,Y -540.741,Z 833.066,A 0.000,B 0.000,C 90.000,E1 47.838} C_DIS
LIN {X -0.043,Y -537.185,Z 833.062,A 0.000,B 0.000,C 90.000,E1 47.148} C_DIS
LIN {X -0.270,Y -533.227,Z 833.058,A 0.000,B 0.000,C 90.000,E1 46.458} C_DIS
LIN {X 0.248,Y -530.730,Z 833.056,A 0.000,B 0.000,C 90.000,E1 45.972} C_DIS
LIN {X 0.165,Y -527.037,Z 833.052,A 0.000,B 0.000,C 90.000,E1 45.405} C_DIS
LIN {X 0.209,Y -521.830,Z 833.048,A 0.000,B 0.000,C 90.000,E1 44.676} C_DIS
LIN {X 0.065,Y -517.317,Z 833.045,A 0.000,B 0.000,C 90.000,E1 44.109} C_DIS
LIN {X 0.020,Y -511.269,Z 833.041,A 0.000,B 0.000,C 90.000,E1 43.380} C_DIS
LIN {X 0.104,Y -507.337,Z 833.039,A 0.000,B 0.000,C 90.000,E1 42.933} C_DIS
LIN {X -0.107,Y -501.016,Z 833.035,A 0.000,B 0.000,C 90.000,E1 42.285} C_DIS
LIN {X 0.009,Y -495.439,Z 833.032,A 0.000,B 0.000,C 90.000,E1 41.714} C_DIS
LIN {X 0.242,Y -489.553,Z 833.029,A 0.000,B 0.000,C 90.000,E1 41.148} C_DIS
LIN {X -0.065,Y -483.526,Z 833.026,A 0.000,B 0.000,C 90.000,E1 40.663} C_DIS
LIN {X 0.186,Y -475.866,Z 833.022,A 0.000,B 0.000,C 90.000,E1 40.011} C_DIS
LIN {X -0.089,Y -466.474,Z 833.018,A 0.000,B 0.000,C 90.000,E1 39.322} C_DIS
LIN {X -0.025,Y -454.082,Z 833.013,A 0.000,B 0.000,C 90.000,E1 38.382} C_DIS
LIN {X -0.053,Y -441.350,Z 833.008,A 0.000,B 0.000,C 90.000,E1 37.443} C_DIS
LIN {X 0.011,Y -419.671,Z 832.999,A 0.000,B 0.000,C 90.000,E1 35.724} C_DIS
LIN {X -0.077,Y -409.134,Z 832.993,A 0.000,B 0.000,C 90.000,E1 34.818} C_DIS
LIN {X -0.027,Y -401.934,Z 832.990,A 0.000,B 0.000,C 90.000,E1 34.119} C_DIS
LIN {X 0.104,Y -397.851,Z 832.987,A 0.000,B 0.000,C 90.000,E1 33.627} C_DIS
LIN {X -0.076,Y -396.036,Z 832.985,A 0.000,B 0.000,C 90.000,E1 33.372} C_DIS
LIN {X -0.114,Y -396.017,Z 832.985,A 0.000,B 0.000,C 90.000,E1 33.372} C_DIS
LIN {X 0.151,Y -394.061,Z 832.978,A 0.000,B 0.000,C 90.000,E1 32.005} C_DIS
LIN {X 0.017,Y -393.489,Z 832.976,A 0.000,B 0.000,C 90.000,E1 31.671} C_DIS
LIN {X 0.140,Y -391.427,Z 832.970,A 0.000,B 0.000,C 90.000,E1 30.590} C_DIS
LIN {X -0.104,Y -391.879,Z 832.962,A 0.000,B 0.000,C 90.000,E1 29.205} C_DIS
LIN {X 0.079,Y -393.249,Z 832.948,A 0.000,B 0.000,C 90.000,E1 26.693} C_DIS
LIN {X 0.132,Y -394.976,Z 832.935,A 0.000,B 0.000,C 90.000,E1 24.207} C_DIS
LIN {X -0.103,Y -396.903,Z 832.921,A 0.000,B 0.000,C 90.000,E1 21.770} C_DIS
LIN {X -0.139,Y -399.470,Z 832.905,A 0.000,B 0.000,C 90.000,E1 18.960} C_DIS
LIN {X 0.196,Y -403.975,Z 832.884,A 0.000,B 0.000,C 90.000,E1 15.064} C_DIS
LIN {X 0.087,Y -407.492,Z 832.870,A 0.000,B 0.000,C 90.000,E1 12.647} C_DIS
LIN {X -0.121,Y -410.845,Z 832.859,A 0.000,B 0.000,C 90.000,E1 10.602} C_DIS
LIN {X 0.127,Y -414.984,Z 832.846,A 0.000,B 0.000,C 90.000,E1 8.163} C_DIS
LIN {X -0.099,Y -418.007,Z 832.836,A 0.000,B 0.000,C 90.000,E1 6.486} C_DIS
LIN {X 0.159,Y -422.382,Z 832.823,A 0.000,B 0.000,C 90.000,E1 4.073} C_DIS
LIN {X 0.181,Y -427.810,Z 832.808,A 0.000,B 0.000,C 90.000,E1 1.375} C_DIS
LIN {X 0.057,Y -434.344,Z 832.792,A 0.000,B 0.000,C 90.000,E1 358.453} C_DIS
LIN {X 0.005,Y -437.499,Z 832.784,A 0.000,B 0.000,C 90.000,E1 357.135} C_DIS
LIN {X -0.151,Y -442.335,Z 832.773,A 0.000,B 0.000,C 90.000,E1 355.179} C_DIS
LIN {X 0.080,Y -446.506,Z 832.764,A 0.000,B 0.000,C 90.000,E1 353.514} C_DIS
LIN {X -0.145,Y -450.107,Z 832.757,A 0.000,B 0.000,C 90.000,E1 352.243} C_DIS
LIN {X 0.112,Y -451.738,Z 832.754,A 0.000,B 0.000,C 90.000,E1 351.724} C_DIS
LIN {X 0.000,Y -453.888,Z 832.751,A 0.000,B 0.000,C 90.000,E1 351.254} C_DIS
LIN {X -0.244,Y -455.776,Z 832.750,A 0.000,B 0.000,C 90.000,E1 350.971} C_DIS
LIN {X 0.121,Y -460.764,Z 832.747,A 0.000,B 0.000,C 90.000,E1 350.387} C_DIS
LIN {X 0.154,Y -467.018,Z 832.744,A 0.000,B 0.000,C 90.000,E1 349.926} C_DIS
LIN {X 0.220,Y -479.572,Z 832.740,A 0.000,B 0.000,C 90.000,E1 349.162} C_DIS
LIN {X 0.194,Y -491.081,Z 832.736,A 0.000,B 0.000,C 90.000,E1 348.465} C_DIS
LIN {X 0.155,Y -495.832,Z 832.734,A 0.000,B 0.000,C 90.000,E1 348.173} C_DIS
LIN {X 0.018,Y -508.602,Z 832.730,A 0.000,B 0.000,C 90.000,E1 347.353} C_DIS
LIN {X 0.155,Y -517.906,Z 832.726,A 0.000,B 0.000,C 90.000,E1 346.700} C_DIS
LIN {X 0.152,Y -528.544,Z 832.722,A 0.000,B 0.000,C 90.000,E1 345.936} C_DIS
LIN {X -0.103,Y -536.056,Z 832.719,A 0.000,B 0.000,C 90.000,E1 345.408} C_DIS
LIN {X 0.112,Y -543.402,Z 832.716,A 0.000,B 0.000,C 90.000,E1 344.810} C_DIS
LIN {X 0.172,Y -550.467,Z 832.712,A 0.000,B 0.000,C 90.000,E1 344.212} C_DIS
LIN {X -0.150,Y -558.627,Z 832.708,A 0.000,B 0.000,C 90.000,E1 343.504} C_DIS
LIN {X 0.166,Y -563.883,Z 832.706,A 0.000,B 0.000,C 90.000,E1 342.960} C_DIS
LIN {X -0.123,Y -567.746,Z 832.703,A 0.000,B 0.000,C 90.000,E1 342.598} C_DIS
LIN {X -0.066,Y -572.645,Z 832.700,A 0.000,B 0.000,C 90.000,E1 342.054} C_DIS
LIN {X 0.118,Y -579.692,Z 832.696,A 0.000,B 0.000,C 90.000,E1 341.221} C_DIS
LIN {X 0.077,Y -584.949,Z 832.692,A 0.000,B 0.000,C 90.000,E1 340.550} C_DIS
LIN {X 0.019,Y -590.717,Z 832.688,A 0.000,B 0.000,C 90.000,E1 339.752} C_DIS
LIN {X 0.024,Y -596.086,Z 832.683,A 0.000,B 0.000,C 90.000,E1 338.954} C_DIS
LIN {X 0.127,Y -600.262,Z 832.679,A 0.000,B 0.000,C 90.000,E1 338.284} C_DIS
LIN {X -0.297,Y -604.147,Z 832.676,A 0.000,B 0.000,C 90.000,E1 337.667} C_DIS
LIN {X -0.216,Y -610.129,Z 832.670,A 0.000,B 0.000,C 90.000,E1 336.613} C_DIS
LIN {X 0.211,Y -615.231,Z 832.665,A 0.000,B 0.000,C 90.000,E1 335.665} C_DIS
LIN {X -0.122,Y -620.698,Z 832.659,A 0.000,B 0.000,C 90.000,E1 334.665} C_DIS
LIN {X -0.130,Y -623.917,Z 832.656,A 0.000,B 0.000,C 90.000,E1 334.024} C_DIS
LIN {X -0.103,Y -627.637,Z 832.651,A 0.000,B 0.000,C 90.000,E1 333.256} C_DIS
LIN {X -0.015,Y -632.247,Z 832.646,A 0.000,B 0.000,C 90.000,E1 332.231} C_DIS
LIN {X -0.079,Y -637.721,Z 832.639,A 0.000,B 0.000,C 90.000,E1 330.973} C_DIS
LIN {X 0.074,Y -640.852,Z 832.635,A 0.000,B 0.000,C 90.000,E1 330.205} C_DIS
LIN {X 0.153,Y -645.839,Z 832.628,A 0.000,B 0.000,C 90.000,E1 328.948} C_DIS
LIN {X -0.324,Y -649.363,Z 832.622,A 0.000,B 0.000,C 90.000,E1 327.995} C_DIS
LIN {X 0.233,Y -653.554,Z 832.615,A 0.000,B 0.000,C 90.000,E1 326.707} C_DIS
LIN {X -0.229,Y -657.328,Z 832.608,A 0.000,B 0.000,C 90.000,E1 325.515} C_DIS
LIN {X -0.120,Y -659.395,Z 832.604,A 0.000,B 0.000,C 90.000,E1 324.769} C_DIS
LIN {X -0.054,Y -661.987,Z 832.599,A 0.000,B 0.000,C 90.000,E1 323.783} C_DIS
LIN {X 0.041,Y -664.254,Z 832.593,A 0.000,B 0.000,C 90.000,E1 322.798} C_DIS
LIN {X 0.043,Y -666.400,Z 832.588,A 0.000,B 0.000,C 90.000,E1 321.823} C_DIS
LIN {X -0.335,Y -668.276,Z 832.583,A 0.000,B 0.000,C 90.000,E1 320.884} C_DIS
LIN {X 0.242,Y -670.444,Z 832.576,A 0.000,B 0.000,C 90.000,E1 319.622} C_DIS
LIN {X -0.172,Y -672.021,Z 832.570,A 0.000,B 0.000,C 90.000,E1 318.690} C_DIS
LIN {X -0.041,Y -673.966,Z 832.564,A 0.000,B 0.000,C 90.000,E1 317.472} C_DIS
LIN {X 0.029,Y -675.018,Z 832.560,A 0.000,B 0.000,C 90.000,E1 316.743} C_DIS
LIN {X -0.193,Y -677.503,Z 832.549,A 0.000,B 0.000,C 90.000,E1 314.838} C_DIS
LIN {X -0.008,Y -678.799,Z 832.542,A 0.000,B 0.000,C 90.000,E1 313.623} C_DIS
LIN {X -0.273,Y -680.153,Z 832.536,A 0.000,B 0.000,C 90.000,E1 312.447} C_DIS
LIN {X -0.013,Y -681.442,Z 832.529,A 0.000,B 0.000,C 90.000,E1 311.229} C_DIS
LIN {X 0.271,Y -682.628,Z 832.522,A 0.000,B 0.000,C 90.000,E1 310.011} C_DIS
LIN {X -0.257,Y -683.909,Z 832.515,A 0.000,B 0.000,C 90.000,E1 308.624} C_DIS
LIN {X 0.203,Y -685.169,Z 832.507,A 0.000,B 0.000,C 90.000,E1 307.156} C_DIS
LIN {X -0.318,Y -686.188,Z 832.500,A 0.000,B 0.000,C 90.000,E1 306.011} C_DIS
LIN {X 0.103,Y -686.926,Z 832.495,A 0.000,B 0.000,C 90.000,E1 305.025} C_DIS
LIN {X -0.209,Y -687.943,Z 832.487,A 0.000,B 0.000,C 90.000,E1 303.627} C_DIS
LIN {X 0.276,Y -689.092,Z 832.478,A 0.000,B 0.000,C 90.000,E1 301.926} C_DIS
LIN {X 0.078,Y -690.349,Z 832.468,A 0.000,B 0.000,C 90.000,E1 300.285} C_DIS
LIN {X -0.110,Y -691.768,Z 832.458,A 0.000,B 0.000,C 90.000,E1 298.409} C_DIS
LIN {X 0.285,Y -693.255,Z 832.447,A 0.000,B 0.000,C 90.000,E1 296.488} C_DIS
LIN {X -0.275,Y -694.058,Z 832.442,A 0.000,B 0.000,C 90.000,E1 295.591} C_DIS
LIN {X 0.049,Y -695.082,Z 832.436,A 0.000,B 0.000,C 90.000,E1 294.387} C_DIS
LIN {X 0.266,Y -695.192,Z 832.433,A 0.000,B 0.000,C 90.000,E1 293.898} C_DIS
LIN {X -0.119,Y -695.153,Z 832.432,A 0.000,B 0.000,C 90.000,E1 293.695} C_DIS
LIN {X 0.103,Y -694.413,Z 832.429,A 0.000,B 0.000,C 90.000,E1 293.206} C_DIS
LIN {X 0.349,Y -693.755,Z 832.428,A 0.000,B 0.000,C 90.000,E1 292.950} C_DIS
LIN {X -0.195,Y -691.655,Z 832.426,A 0.000,B 0.000,C 90.000,E1 292.642} C_DIS
LIN {X 0.041,Y -690.092,Z 832.424,A 0.000,B 0.000,C 90.000,E1 292.386} C_DIS
LIN {X -0.105,Y -688.969,Z 832.424,A 0.000,B 0.000,C 90.000,E1 292.280} C_DIS
LIN {X 0.122,Y -685.552,Z 832.422,A 0.000,B 0.000,C 90.000,E1 292.025} C_DIS
LIN {X -0.012,Y -682.148,Z 832.421,A 0.000,B 0.000,C 90.000,E1 291.844} C_DIS
LIN {X -0.130,Y -680.472,Z 832.421,A 0.000,B 0.000,C 90.000,E1 291.770} C_DIS
LIN {X -0.259,Y -672.346,Z 832.420,A 0.000,B 0.000,C 90.000,E1 291.535} C_DIS
LIN {X 0.234,Y -665.993,Z 832.419,A 0.000,B 0.000,C 90.000,E1 291.354} C_DIS
LIN {X -0.121,Y -659.936,Z 832.418,A 0.000,B 0.000,C 90.000,E1 291.280} C_DIS
LIN {X -0.074,Y -649.861,Z 832.417,A 0.000,B 0.000,C 90.000,E1 291.099} C_DIS
LIN {X 0.022,Y -641.992,Z 832.416,A 0.000,B 0.000,C 90.000,E1 290.918} C_DIS
LIN {X -0.292,Y -634.230,Z 832.415,A 0.000,B 0.000,C 90.000,E1 290.737} C_DIS
LIN {X -0.275,Y -630.669,Z 832.414,A 0.000,B 0.000,C 90.000,E1 290.610} C_DIS
LIN {X -0.110,Y -625.333,Z 832.413,A 0.000,B 0.000,C 90.000,E1 290.355} C_DIS
LIN {X 0.169,Y -622.802,Z 832.412,A 0.000,B 0.000,C 90.000,E1 290.174} C_DIS
LIN {X 0.258,Y -621.650,Z 832.412,A 0.000,B 0.000,C 90.000,E1 290.066} C_DIS
LIN {X 0.041,Y -621.056,Z 832.411,A 0.000,B 0.000,C 90.000,E1 289.939} C_DIS
LIN {X -0.253,Y -621.483,Z 832.410,A 0.000,B 0.000,C 90.000,E1 289.758} C_DIS
LIN {X -0.197,Y -623.200,Z 832.407,A 0.000,B 0.000,C 90.000,E1 289.322} C_DIS
LIN {X 0.157,Y -625.316,Z 832.405,A 0.000,B 0.000,C 90.000,E1 288.906} C_DIS
LIN {X -0.203,Y -629.867,Z 832.401,A 0.000,B 0.000,C 90.000,E1 288.181} C_DIS
LIN {X 0.000,Y -634.211,Z 832.396,A 0.000,B 0.000,C 90.000,E1 287.275} C_DIS
LIN {X -0.370,Y -636.421,Z 832.393,A 0.000,B 0.000,C 90.000,E1 286.804} C_DIS
LIN {X 0.069,Y -638.352,Z 832.390,A 0.000,B 0.000,C 90.000,E1 286.260} C_DIS
LIN {X 0.355,Y -640.922,Z 832.386,A 0.000,B 0.000,C 90.000,E1 285.481} C_DIS
LIN {X -0.125,Y -642.866,Z 832.382,A 0.000,B 0.000,C 90.000,E1 284.773} C_DIS
LIN {X 0.192,Y -644.032,Z 832.379,A 0.000,B 0.000,C 90.000,E1 284.245} C_DIS
LIN {X -0.254,Y -645.190,Z 832.375,A 0.000,B 0.000,C 90.000,E1 283.536} C_DIS
LIN {X 0.083,Y -645.766,Z 832.372,A 0.000,B 0.000,C 90.000,E1 283.008} C_DIS
LIN {X -0.205,Y -645.989,Z 832.370,A 0.000,B 0.000,C 90.000,E1 282.535} C_DIS
LIN {X -0.007,Y -645.698,Z 832.365,A 0.000,B 0.000,C 90.000,E1 281.771} C_DIS
LIN {X 0.332,Y -645.324,Z 832.363,A 0.000,B 0.000,C 90.000,E1 281.243} C_DIS
LIN {X -0.086,Y -644.626,Z 832.360,A 0.000,B 0.000,C 90.000,E1 280.782} C_DIS
LIN {X 0.244,Y -643.652,Z 832.357,A 0.000,B 0.000,C 90.000,E1 280.254} C_DIS
LIN {X -0.177,Y -642.417,Z 832.354,A 0.000,B 0.000,C 90.000,E1 279.792} C_DIS
LIN {X -0.336,Y -641.719,Z 832.353,A 0.000,B 0.000,C 90.000,E1 279.557} C_DIS
LIN {X -0.031,Y -639.937,Z 832.350,A 0.000,B 0.000,C 90.000,E1 279.029} C_DIS
LIN {X 0.025,Y -637.125,Z 832.347,A 0.000,B 0.000,C 90.000,E1 278.398} C_DIS
LIN {X 0.286,Y -634.376,Z 832.344,A 0.000,B 0.000,C 90.000,E1 277.871} C_DIS
LIN {X -0.189,Y -631.059,Z 832.341,A 0.000,B 0.000,C 90.000,E1 277.409} C_DIS
LIN {X -0.058,Y -627.304,Z 832.338,A 0.000,B 0.000,C 90.000,E1 276.891} C_DIS
LIN {X -0.101,Y -621.413,Z 832.335,A 0.000,B 0.000,C 90.000,E1 276.258} C_DIS
LIN {X -0.252,Y -615.726,Z 832.332,A 0.000,B 0.000,C 90.000,E1 275.796} C_DIS
LIN {X -0.282,Y -612.557,Z 832.331,A 0.000,B 0.000,C 90.000,E1 275.568} C_DIS
LIN {X -0.142,Y -606.074,Z 832.329,A 0.000,B 0.000,C 90.000,E1 275.163} C_DIS
LIN {X 0.262,Y -597.198,Z 832.326,A 0.000,B 0.000,C 90.000,E1 274.702} C_DIS
LIN {X 0.229,Y -591.855,Z 832.325,A 0.000,B 0.000,C 90.000,E1 274.473} C_DIS
LIN {X -0.245,Y -584.737,Z 832.323,A 0.000,B 0.000,C 90.000,E1 274.245} C_DIS
LIN {X 0.280,Y -578.978,Z 832.323,A 0.000,B 0.000,C 90.000,E1 274.012} C_DIS
LIN {X 0.037,Y -572.481,Z 832.322,A 0.000,B 0.000,C 90.000,E1 273.898} C_DIS
LIN {X -0.199,Y -565.074,Z 832.321,A 0.000,B 0.000,C 90.000,E1 273.841} C_DIS
LIN {X 0.191,Y -559.205,Z 832.321,A 0.000,B 0.000,C 90.000,E1 273.784} C_DIS
LIN {X 0.134,Y -554.921,Z 832.321,A 0.000,B 0.000,C 90.000,E1 273.784} C_DIS
LIN {X 0.022,Y -553.093,Z 832.321,A 0.000,B 0.000,C 90.000,E1 273.784} C_DIS
LIN {X -0.084,Y -550.453,Z 832.321,A 0.000,B 0.000,C 90.000,E1 273.726} C_DIS
LIN {X -0.139,Y -550.364,Z 832.321,A 0.000,B 0.000,C 90.000,E1 273.726} C_DIS
LIN {X 0.076,Y -549.484,Z 832.319,A 0.000,B 0.000,C 90.000,E1 273.383} C_DIS
LIN {X 0.157,Y -548.884,Z 832.317,A 0.000,B 0.000,C 90.000,E1 273.094} C_DIS
LIN {X 0.132,Y -546.631,Z 832.305,A 0.000,B 0.000,C 90.000,E1 270.859} C_DIS
LIN {X -0.120,Y -545.207,Z 832.294,A 0.000,B 0.000,C 90.000,E1 268.912} C_DIS
LIN {X 0.078,Y -544.219,Z 832.286,A 0.000,B 0.000,C 90.000,E1 267.478} C_DIS
LIN {X -0.222,Y -543.087,Z 832.277,A 0.000,B 0.000,C 90.000,E1 265.812} C_DIS
LIN {X -0.010,Y -541.977,Z 832.267,A 0.000,B 0.000,C 90.000,E1 264.090} C_DIS
LIN {X 0.213,Y -540.873,Z 832.259,A 0.000,B 0.000,C 90.000,E1 262.648} C_DIS
LIN {X 0.010,Y -538.996,Z 832.248,A 0.000,B 0.000,C 90.000,E1 260.679} C_DIS
LIN {X 0.215,Y -538.174,Z 832.244,A 0.000,B 0.000,C 90.000,E1 259.803} C_DIS
LIN {X -0.091,Y -536.757,Z 832.236,A 0.000,B 0.000,C 90.000,E1 258.409} C_DIS
LIN {X -0.094,Y -534.732,Z 832.224,A 0.000,B 0.000,C 90.000,E1 256.408} C_DIS
LIN {X -0.015,Y -532.448,Z 832.213,A 0.000,B 0.000,C 90.000,E1 254.393} C_DIS
LIN {X -0.058,Y -530.801,Z 832.205,A 0.000,B 0.000,C 90.000,E1 252.960} C_DIS
LIN {X 0.039,Y -528.676,Z 832.196,A 0.000,B 0.000,C 90.000,E1 251.221} C_DIS
LIN {X 0.079,Y -527.171,Z 832.189,A 0.000,B 0.000,C 90.000,E1 250.061} C_DIS
LIN {X 0.270,Y -525.120,Z 832.181,A 0.000,B 0.000,C 90.000,E1 248.592} C_DIS
LIN {X 0.089,Y -522.664,Z 832.172,A 0.000,B 0.000,C 90.000,E1 246.869} C_DIS
LIN {X -0.247,Y -520.871,Z 832.165,A 0.000,B 0.000,C 90.000,E1 245.741} C_DIS
LIN {X -0.248,Y -518.571,Z 832.157,A 0.000,B 0.000,C 90.000,E1 244.280} C_DIS
LIN {X 0.045,Y -516.584,Z 832.151,A 0.000,B 0.000,C 90.000,E1 243.076} C_DIS
LIN {X 0.092,Y -513.451,Z 832.141,A 0.000,B 0.000,C 90.000,E1 241.307} C_DIS
LIN {X 0.089,Y -511.334,Z 832.134,A 0.000,B 0.000,C 90.000,E1 240.127} C_DIS
LIN {X -0.052,Y -508.585,Z 832.126,A 0.000,B 0.000,C 90.000,E1 238.663} C_DIS
LIN {X 0.128,Y -506.262,Z 832.119,A 0.000,B 0.000,C 90.000,E1 237.454} C_DIS
LIN {X 0.152,Y -503.141,Z 832.111,A 0.000,B 0.000,C 90.000,E1 235.960} C_DIS
LIN {X 0.101,Y -500.445,Z 832.104,A 0.000,B 0.000,C 90.000,E1 234.769} C_DIS
LIN {X -0.119,Y -496.945,Z 832.096,A 0.000,B 0.000,C 90.000,E1 233.290} C_DIS
LIN {X 0.195,Y -493.406,Z 832.088,A 0.000,B 0.000,C 90.000,E1 231.743} C_DIS
LIN {X 0.275,Y -487.679,Z 832.074,A 0.000,B 0.000,C 90.000,E1 229.299} C_DIS
LIN {X 0.222,Y -484.835,Z 832.067,A 0.000,B 0.000,C 90.000,E1 228.081} C_DIS
LIN {X -0.170,Y -479.984,Z 832.055,A 0.000,B 0.000,C 90.000,E1 225.972} C_DIS
LIN {X -0.022,Y -477.244,Z 832.048,A 0.000,B 0.000,C 90.000,E1 224.717} C_DIS
LIN {X -0.131,Y -475.957,Z 832.045,A 0.000,B 0.000,C 90.000,E1 224.109} C_DIS
LIN {X 0.011,Y -470.632,Z 832.031,A 0.000,B 0.000,C 90.000,E1 221.595} C_DIS
LIN {X -0.046,Y -465.975,Z 832.019,A 0.000,B 0.000,C 90.000,E1 219.402} C_DIS
LIN {X 0.199,Y -461.380,Z 832.007,A 0.000,B 0.000,C 90.000,E1 217.156} C_DIS
LIN {X 0.193,Y -458.730,Z 832.000,A 0.000,B 0.000,C 90.000,E1 215.884} C_DIS
LIN {X -0.123,Y -455.407,Z 831.991,A 0.000,B 0.000,C 90.000,E1 214.326} C_DIS
LIN {X -0.005,Y -451.918,Z 831.982,A 0.000,B 0.000,C 90.000,E1 212.704} C_DIS
LIN {X 0.054,Y -448.546,Z 831.973,A 0.000,B 0.000,C 90.000,E1 211.082} C_DIS
LIN {X -0.054,Y -443.929,Z 831.960,A 0.000,B 0.000,C 90.000,E1 208.821} C_DIS
LIN {X -0.128,Y -439.439,Z 831.947,A 0.000,B 0.000,C 90.000,E1 206.539} C_DIS
LIN {X 0.236,Y -435.411,Z 831.936,A 0.000,B 0.000,C 90.000,E1 204.515} C_DIS
LIN {X -0.241,Y -431.364,Z 831.925,A 0.000,B 0.000,C 90.000,E1 202.589} C_DIS
LIN {X -0.212,Y -428.192,Z 831.916,A 0.000,B 0.000,C 90.000,E1 200.918} C_DIS
LIN {X -0.001,Y -424.931,Z 831.907,A 0.000,B 0.000,C 90.000,E1 199.214} C_DIS
LIN {X 0.137,Y -421.605,Z 831.897,A 0.000,B 0.000,C 90.000,E1 197.511} C_DIS
LIN {X -0.048,Y -418.416,Z 831.888,A 0.000,B 0.000,C 90.000,E1 195.843} C_DIS
LIN {X 0.109,Y -415.182,Z 831.879,A 0.000,B 0.000,C 90.000,E1 194.120} C_DIS
LIN {X 0.126,Y -411.119,Z 831.867,A 0.000,B 0.000,C 90.000,E1 192.063} C_DIS
LIN {X -0.039,Y -407.160,Z 831.856,A 0.000,B 0.000,C 90.000,E1 190.018} C_DIS
LIN {X -0.030,Y -403.252,Z 831.844,A 0.000,B 0.000,C 90.000,E1 187.936} C_DIS
LIN {X -0.100,Y -399.941,Z 831.834,A 0.000,B 0.000,C 90.000,E1 186.201} C_DIS
LIN {X -0.053,Y -395.044,Z 831.819,A 0.000,B 0.000,C 90.000,E1 183.383} C_DIS
LIN {X 0.023,Y -390.011,Z 831.799,A 0.000,B 0.000,C 90.000,E1 179.828} C_DIS
LIN {X 0.064,Y -388.221,Z 831.791,A 0.000,B 0.000,C 90.000,E1 178.396} C_DIS
LIN {X -0.099,Y -385.534,Z 831.779,A 0.000,B 0.000,C 90.000,E1 176.274} C_DIS
LIN {X 0.082,Y -382.862,Z 831.767,A 0.000,B 0.000,C 90.000,E1 174.090} C_DIS
LIN {X 0.186,Y -379.997,Z 831.753,A 0.000,B 0.000,C 90.000,E1 171.546} C_DIS
LIN {X 0.093,Y -378.240,Z 831.743,A 0.000,B 0.000,C 90.000,E1 169.746} C_DIS
LIN {X 0.030,Y -376.510,Z 831.733,A 0.000,B 0.000,C 90.000,E1 167.937} C_DIS
LIN {X -0.167,Y -374.134,Z 831.717,A 0.000,B 0.000,C 90.000,E1 165.046} C_DIS
LIN {X -0.073,Y -372.920,Z 831.705,A 0.000,B 0.000,C 90.000,E1 162.834} C_DIS
LIN {X 0.107,Y -372.370,Z 831.692,A 0.000,B 0.000,C 90.000,E1 160.604} C_DIS
LIN {X 0.043,Y -372.910,Z 831.680,A 0.000,B 0.000,C 90.000,E1 158.411} C_DIS
LIN {X 0.113,Y -373.327,Z 831.676,A 0.000,B 0.000,C 90.000,E1 157.667} C_DIS
LIN {X 0.187,Y -373.923,Z 831.672,A 0.000,B 0.000,C 90.000,E1 156.922} C_DIS
LIN {X -0.076,Y -374.729,Z 831.668,A 0.000,B 0.000,C 90.000,E1 156.230} C_DIS
LIN {X 0.131,Y -376.469,Z 831.662,A 0.000,B 0.000,C 90.000,E1 155.101} C_DIS
LIN {X 0.034,Y -378.539,Z 831.657,A 0.000,B 0.000,C 90.000,E1 154.204} C_DIS
LIN {X -0.197,Y -380.705,Z 831.653,A 0.000,B 0.000,C 90.000,E1 153.512} C_DIS
LIN {X -0.064,Y -382.615,Z 831.650,A 0.000,B 0.000,C 90.000,E1 152.948} C_DIS
LIN {X -0.083,Y -385.129,Z 831.647,A 0.000,B 0.000,C 90.000,E1 152.410} C_DIS
LIN {X 0.160,Y -389.918,Z 831.643,A 0.000,B 0.000,C 90.000,E1 151.641} C_DIS
LIN {X -0.223,Y -393.651,Z 831.640,A 0.000,B 0.000,C 90.000,E1 151.257} C_DIS
LIN {X 0.036,Y -395.399,Z 831.639,A 0.000,B 0.000,C 90.000,E1 151.051} C_DIS
LIN {X 0.223,Y -401.106,Z 831.637,A 0.000,B 0.000,C 90.000,E1 150.589} C_DIS
LIN {X -0.049,Y -402.898,Z 831.636,A 0.000,B 0.000,C 90.000,E1 150.511} C_DIS
LIN {X -0.065,Y -412.260,Z 831.634,A 0.000,B 0.000,C 90.000,E1 150.049} C_DIS
LIN {X 0.018,Y -418.703,Z 831.632,A 0.000,B 0.000,C 90.000,E1 149.744} C_DIS
LIN {X 0.015,Y -425.745,Z 831.630,A 0.000,B 0.000,C 90.000,E1 149.410} C_DIS
LIN {X 0.061,Y -435.297,Z 831.627,A 0.000,B 0.000,C 90.000,E1 148.869} C_DIS
LIN {X 0.158,Y -438.363,Z 831.626,A 0.000,B 0.000,C 90.000,E1 148.663} C_DIS
LIN {X -0.077,Y -449.482,Z 831.622,A 0.000,B 0.000,C 90.000,E1 147.916} C_DIS
LIN {X -0.254,Y -455.353,Z 831.619,A 0.000,B 0.000,C 90.000,E1 147.454} C_DIS
LIN {X -0.097,Y -464.079,Z 831.615,A 0.000,B 0.000,C 90.000,E1 146.628} C_DIS
LIN {X -0.132,Y -468.251,Z 831.612,A 0.000,B 0.000,C 90.000,E1 146.215} C_DIS
LIN {X 0.002,Y -476.378,Z 831.607,A 0.000,B 0.000,C 90.000,E1 145.341} C_DIS
LIN {X 0.043,Y -481.253,Z 831.604,A 0.000,B 0.000,C 90.000,E1 144.769} C_DIS
LIN {X -0.043,Y -489.565,Z 831.598,A 0.000,B 0.000,C 90.000,E1 143.703} C_DIS
LIN {X -0.044,Y -497.065,Z 831.592,A 0.000,B 0.000,C 90.000,E1 142.637} C_DIS
LIN {X -0.249,Y -505.036,Z 831.586,A 0.000,B 0.000,C 90.000,E1 141.457} C_DIS
LIN {X 0.250,Y -508.725,Z 831.582,A 0.000,B 0.000,C 90.000,E1 140.803} C_DIS
LIN {X -0.175,Y -515.671,Z 831.576,A 0.000,B 0.000,C 90.000,E1 139.666} C_DIS
LIN {X -0.186,Y -519.903,Z 831.572,A 0.000,B 0.000,C 90.000,E1 138.933} C_DIS
LIN {X 0.045,Y -526.938,Z 831.565,A 0.000,B 0.000,C 90.000,E1 137.595} C_DIS
LIN {X -0.130,Y -532.858,Z 831.558,A 0.000,B 0.000,C 90.000,E1 136.458} C_DIS
LIN {X -0.075,Y -540.973,Z 831.549,A 0.000,B 0.000,C 90.000,E1 134.879} C_DIS
LIN {X 0.316,Y -546.655,Z 831.543,A 0.000,B 0.000,C 90.000,E1 133.704} C_DIS
LIN {X -0.029,Y -549.377,Z 831.540,A 0.000,B 0.000,C 90.000,E1 133.176} C_DIS
LIN {X -0.209,Y -556.888,Z 831.531,A 0.000,B 0.000,C 90.000,E1 131.515} C_DIS
LIN {X 0.162,Y -559.902,Z 831.527,A 0.000,B 0.000,C 90.000,E1 130.782} C_DIS
LIN {X 0.127,Y -565.337,Z 831.519,A 0.000,B 0.000,C 90.000,E1 129.402} C_DIS
LIN {X 0.017,Y -568.410,Z 831.514,A 0.000,B 0.000,C 90.000,E1 128.588} C_DIS
LIN {X 0.038,Y -571.165,Z 831.510,A 0.000,B 0.000,C 90.000,E1 127.764} C_DIS
LIN {X -0.009,Y -573.684,Z 831.505,A 0.000,B 0.000,C 90.000,E1 126.950} C_DIS
LIN {X 0.280,Y -575.203,Z 831.502,A 0.000,B 0.000,C 90.000,E1 126.377} C_DIS
LIN {X -0.227,Y -576.476,Z 831.499,A 0.000,B 0.000,C 90.000,E1 125.884} C_DIS
LIN {X 0.080,Y -577.600,Z 831.496,A 0.000,B 0.000,C 90.000,E1 125.311} C_DIS
LIN {X -0.095,Y -579.508,Z 831.490,A 0.000,B 0.000,C 90.000,E1 124.246} C_DIS
LIN {X 0.065,Y -580.695,Z 831.486,A 0.000,B 0.000,C 90.000,E1 123.420} C_DIS
LIN {X -0.077,Y -581.664,Z 831.481,A 0.000,B 0.000,C 90.000,E1 122.625} C_DIS
LIN {X -0.057,Y -582.250,Z 831.478,A 0.000,B 0.000,C 90.000,E1 122.084} C_DIS
LIN {X 0.155,Y -582.960,Z 831.471,A 0.000,B 0.000,C 90.000,E1 120.718} C_DIS
LIN {X -0.222,Y -582.924,Z 831.463,A 0.000,B 0.000,C 90.000,E1 119.411} C_DIS
LIN {X 0.179,Y -582.498,Z 831.459,A 0.000,B 0.000,C 90.000,E1 118.565} C_DIS
LIN {X 0.194,Y -582.212,Z 831.456,A 0.000,B 0.000,C 90.000,E1 118.025} C_DIS
LIN {X -0.070,Y -581.630,Z 831.453,A 0.000,B 0.000,C 90.000,E1 117.513} C_DIS
LIN {X 0.051,Y -580.706,Z 831.448,A 0.000,B 0.000,C 90.000,E1 116.693} C_DIS
LIN {X -0.100,Y -579.513,Z 831.444,A 0.000,B 0.000,C 90.000,E1 115.899} C_DIS
LIN {X 0.141,Y -578.479,Z 831.441,A 0.000,B 0.000,C 90.000,E1 115.335} C_DIS
LIN {X -0.145,Y -576.925,Z 831.438,A 0.000,B 0.000,C 90.000,E1 114.823} C_DIS
LIN {X 0.230,Y -575.993,Z 831.436,A 0.000,B 0.000,C 90.000,E1 114.515} C_DIS
LIN {X 0.003,Y -574.308,Z 831.434,A 0.000,B 0.000,C 90.000,E1 114.131} C_DIS
LIN {X -0.023,Y -571.348,Z 831.431,A 0.000,B 0.000,C 90.000,E1 113.590} C_DIS
LIN {X -0.016,Y -566.526,Z 831.427,A 0.000,B 0.000,C 90.000,E1 112.770} C_DIS
LIN {X -0.200,Y -564.940,Z 831.425,A 0.000,B 0.000,C 90.000,E1 112.514} C_DIS
LIN {X -0.111,Y -563.806,Z 831.424,A 0.000,B 0.000,C 90.000,E1 112.333} C_DIS
LIN {X 0.034,Y -563.512,Z 831.423,A 0.000,B 0.000,C 90.000,E1 112.078} C_DIS
LIN {X -0.122,Y -563.296,Z 831.422,A 0.000,B 0.000,C 90.000,E1 112.025} C_DIS
LIN {X 0.147,Y -563.166,Z 831.421,A 0.000,B 0.000,C 90.000,E1 111.791} C_DIS
LIN {X -0.255,Y -563.127,Z 831.418,A 0.000,B 0.000,C 90.000,E1 111.280} C_DIS
LIN {X -0.101,Y -562.825,Z 831.410,A 0.000,B 0.000,C 90.000,E1 109.885} C_DIS
LIN {X -0.165,Y -562.232,Z 831.401,A 0.000,B 0.000,C 90.000,E1 108.236} C_DIS
LIN {X 0.068,Y -562.510,Z 831.383,A 0.000,B 0.000,C 90.000,E1 104.898} C_DIS
LIN {X 0.108,Y -563.665,Z 831.369,A 0.000,B 0.000,C 90.000,E1 102.411} C_DIS
LIN {X 0.205,Y -565.135,Z 831.357,A 0.000,B 0.000,C 90.000,E1 100.197} C_DIS
LIN {X 0.226,Y -565.957,Z 831.351,A 0.000,B 0.000,C 90.000,E1 99.095} C_DIS
LIN {X -0.133,Y -566.898,Z 831.343,A 0.000,B 0.000,C 90.000,E1 97.757} C_DIS
LIN {X 0.271,Y -568.044,Z 831.332,A 0.000,B 0.000,C 90.000,E1 95.796} C_DIS
LIN {X -0.081,Y -568.801,Z 831.323,A 0.000,B 0.000,C 90.000,E1 94.188} C_DIS
LIN {X 0.026,Y -569.333,Z 831.316,A 0.000,B 0.000,C 90.000,E1 92.808} C_DIS
LIN {X -0.207,Y -569.960,Z 831.305,A 0.000,B 0.000,C 90.000,E1 90.917} C_DIS
LIN {X -0.126,Y -570.309,Z 831.297,A 0.000,B 0.000,C 90.000,E1 89.542} C_DIS
LIN {X -0.024,Y -570.679,Z 831.290,A 0.000,B 0.000,C 90.000,E1 88.165} C_DIS
LIN {X -0.223,Y -571.052,Z 831.279,A 0.000,B 0.000,C 90.000,E1 86.274} C_DIS
LIN {X -0.075,Y -571.269,Z 831.272,A 0.000,B 0.000,C 90.000,E1 84.894} C_DIS
LIN {X -0.127,Y -571.690,Z 831.261,A 0.000,B 0.000,C 90.000,E1 82.989} C_DIS
LIN {X 0.022,Y -572.167,Z 831.249,A 0.000,B 0.000,C 90.000,E1 80.792} C_DIS
LIN {X -0.230,Y -572.620,Z 831.241,A 0.000,B 0.000,C 90.000,E1 79.454} C_DIS
LIN {X -0.163,Y -573.157,Z 831.232,A 0.000,B 0.000,C 90.000,E1 77.813} C_DIS
LIN {X 0.108,Y -573.530,Z 831.222,A 0.000,B 0.000,C 90.000,E1 75.880} C_DIS
LIN {X 0.118,Y -573.708,Z 831.214,A 0.000,B 0.000,C 90.000,E1 74.519} C_DIS
LIN {X 0.280,Y -573.724,Z 831.204,A 0.000,B 0.000,C 90.000,E1 72.598} C_DIS
LIN {X -0.095,Y -573.649,Z 831.196,A 0.000,B 0.000,C 90.000,E1 71.275} C_DIS
LIN {X -0.294,Y -573.405,Z 831.185,A 0.000,B 0.000,C 90.000,E1 69.390} C_DIS
LIN {X -0.116,Y -573.179,Z 831.179,A 0.000,B 0.000,C 90.000,E1 68.284} C_DIS
LIN {X 0.056,Y -572.916,Z 831.173,A 0.000,B 0.000,C 90.000,E1 67.177} C_DIS
LIN {X 0.281,Y -572.508,Z 831.166,A 0.000,B 0.000,C 90.000,E1 65.793} C_DIS
LIN {X 0.147,Y -572.113,Z 831.160,A 0.000,B 0.000,C 90.000,E1 64.717} C_DIS
LIN {X -0.159,Y -571.521,Z 831.152,A 0.000,B 0.000,C 90.000,E1 63.384} C_DIS
LIN {X 0.115,Y -570.588,Z 831.143,A 0.000,B 0.000,C 90.000,E1 61.719} C_DIS
LIN {X 0.047,Y -570.290,Z 831.140,A 0.000,B 0.000,C 90.000,E1 61.179} C_DIS
LIN {X 0.130,Y -569.290,Z 831.134,A 0.000,B 0.000,C 90.000,E1 60.078} C_DIS
LIN {X -0.193,Y -567.834,Z 831.126,A 0.000,B 0.000,C 90.000,E1 58.742} C_DIS
LIN {X -0.239,Y -566.120,Z 831.119,A 0.000,B 0.000,C 90.000,E1 57.375} C_DIS
LIN {X 0.363,Y -564.482,Z 831.113,A 0.000,B 0.000,C 90.000,E1 56.215} C_DIS
LIN {X -0.098,Y -563.099,Z 831.108,A 0.000,B 0.000,C 90.000,E1 55.435} C_DIS
LIN {X -0.108,Y -561.524,Z 831.103,A 0.000,B 0.000,C 90.000,E1 54.609} C_DIS
LIN {X -0.048,Y -559.171,Z 831.097,A 0.000,B 0.000,C 90.000,E1 53.497} C_DIS
LIN {X 0.220,Y -557.171,Z 831.093,A 0.000,B 0.000,C 90.000,E1 52.637} C_DIS
LIN {X 0.025,Y -554.908,Z 831.088,A 0.000,B 0.000,C 90.000,E1 51.823} C_DIS
LIN {X 0.173,Y -553.265,Z 831.085,A 0.000,B 0.000,C 90.000,E1 51.251} C_DIS
LIN {X -0.120,Y -551.531,Z 831.082,A 0.000,B 0.000,C 90.000,E1 50.723} C_DIS
LIN {X 0.052,Y -548.589,Z 831.077,A 0.000,B 0.000,C 90.000,E1 49.865} C_DIS
LIN {X 0.084,Y -546.493,Z 831.074,A 0.000,B 0.000,C 90.000,E1 49.299} C_DIS
LIN {X -0.221,Y -542.915,Z 831.069,A 0.000,B 0.000,C 90.000,E1 48.485} C_DIS
LIN {X -0.219,Y -540.354,Z 831.066,A 0.000,B 0.000,C 90.000,E1 47.919} C_DIS
LIN {X 0.161,Y -537.536,Z 831.063,A 0.000,B 0.000,C 90.000,E1 47.310} C_DIS
LIN {X -0.066,Y -533.584,Z 831.059,A 0.000,B 0.000,C 90.000,E1 46.620} C_DIS
LIN {X -0.129,Y -530.173,Z 831.056,A 0.000,B 0.000,C 90.000,E1 46.053} C_DIS
LIN {X -0.213,Y -526.430,Z 831.053,A 0.000,B 0.000,C 90.000,E1 45.486} C_DIS
LIN {X 0.047,Y -522.273,Z 831.049,A 0.000,B 0.000,C 90.000,E1 44.879} C_DIS
LIN {X -0.008,Y -517.860,Z 831.046,A 0.000,B 0.000,C 90.000,E1 44.312} C_DIS
LIN {X -0.018,Y -513.145,Z 831.043,A 0.000,B 0.000,C 90.000,E1 43.743} C_DIS
LIN {X -0.004,Y -509.745,Z 831.041,A 0.000,B 0.000,C 90.000,E1 43.338} C_DIS
LIN {X 0.042,Y -502.976,Z 831.037,A 0.000,B 0.000,C 90.000,E1 42.609} C_DIS
LIN {X -0.021,Y -496.063,Z 831.033,A 0.000,B 0.000,C 90.000,E1 41.919} C_DIS
LIN {X 0.140,Y -488.697,Z 831.029,A 0.000,B 0.000,C 90.000,E1 41.229} C_DIS
LIN {X -0.065,Y -484.150,Z 831.027,A 0.000,B 0.000,C 90.000,E1 40.862} C_DIS
LIN {X -0.140,Y -476.528,Z 831.024,A 0.000,B 0.000,C 90.000,E1 40.253} C_DIS
LIN {X -0.076,Y -468.781,Z 831.020,A 0.000,B 0.000,C 90.000,E1 39.644} C_DIS
LIN {X 0.155,Y -456.143,Z 831.015,A 0.000,B 0.000,C 90.000,E1 38.669} C_DIS
LIN {X -0.093,Y -441.876,Z 831.009,A 0.000,B 0.000,C 90.000,E1 37.649} C_DIS
LIN {X 0.007,Y -418.637,Z 830.999,A 0.000,B 0.000,C 90.000,E1 35.804} C_DIS
LIN {X 0.060,Y -406.671,Z 830.993,A 0.000,B 0.000,C 90.000,E1 34.739} C_DIS
LIN {X 0.054,Y -402.384,Z 830.991,A 0.000,B 0.000,C 90.000,E1 34.326} C_DIS
LIN {X 0.123,Y -397.896,Z 830.988,A 0.000,B 0.000,C 90.000,E1 33.785} C_DIS
LIN {X 0.071,Y -396.396,Z 830.987,A 0.000,B 0.000,C 90.000,E1 33.579} C_DIS
LIN {X 0.048,Y -396.379,Z 830.987,A 0.000,B 0.000,C 90.000,E1 33.579} C_DIS
LIN {X 0.024,Y -394.036,Z 830.978,A 0.000,B 0.000,C 90.000,E1 32.005} C_DIS
LIN {X -0.246,Y -392.748,Z 830.974,A 0.000,B 0.000,C 90.000,E1 31.337} C_DIS
LIN {X 0.083,Y -391.559,Z 830.971,A 0.000,B 0.000,C 90.000,E1 30.669} C_DIS
LIN {X -0.070,Y -393.277,Z 830.950,A 0.000,B 0.000,C 90.000,E1 27.052} C_DIS
LIN {X 0.017,Y -395.205,Z 830.935,A 0.000,B 0.000,C 90.000,E1 24.207} C_DIS
LIN {X 0.156,Y -397.110,Z 830.921,A 0.000,B 0.000,C 90.000,E1 21.716} C_DIS
LIN {X 0.135,Y -399.666,Z 830.905,A 0.000,B 0.000,C 90.000,E1 18.906} C_DIS
LIN {X 0.101,Y -404.175,Z 830.884,A 0.000,B 0.000,C 90.000,E1 15.064} C_DIS
LIN {X -0.104,Y -407.170,Z 830.872,A 0.000,B 0.000,C 90.000,E1 13.008} C_DIS
LIN {X 0.196,Y -411.074,Z 830.859,A 0.000,B 0.000,C 90.000,E1 10.546} C_DIS
LIN {X 0.047,Y -415.243,Z 830.845,A 0.000,B 0.000,C 90.000,E1 8.163} C_DIS
LIN {X 0.187,Y -417.648,Z 830.838,A 0.000,B 0.000,C 90.000,E1 6.777} C_DIS
LIN {X 0.028,Y -421.365,Z 830.827,A 0.000,B 0.000,C 90.000,E1 4.759} C_DIS
LIN {X -0.013,Y -426.642,Z 830.812,A 0.000,B 0.000,C 90.000,E1 2.064} C_DIS
LIN {X 0.000,Y -431.025,Z 830.800,A 0.000,B 0.000,C 90.000,E1 360.000} C_DIS
LIN {X -0.085,Y -436.942,Z 830.786,A 0.000,B 0.000,C 90.000,E1 357.478} C_DIS
LIN {X -0.140,Y -442.530,Z 830.773,A 0.000,B 0.000,C 90.000,E1 355.179} C_DIS
LIN {X 0.095,Y -446.672,Z 830.764,A 0.000,B 0.000,C 90.000,E1 353.514} C_DIS
LIN {X -0.127,Y -450.169,Z 830.757,A 0.000,B 0.000,C 90.000,E1 352.243} C_DIS
LIN {X -0.185,Y -452.332,Z 830.753,A 0.000,B 0.000,C 90.000,E1 351.602} C_DIS
LIN {X 0.087,Y -454.449,Z 830.751,A 0.000,B 0.000,C 90.000,E1 351.084} C_DIS
LIN {X 0.156,Y -455.327,Z 830.750,A 0.000,B 0.000,C 90.000,E1 350.914} C_DIS
LIN {X 0.017,Y -458.594,Z 830.748,A 0.000,B 0.000,C 90.000,E1 350.557} C_DIS
LIN {X -0.003,Y -460.399,Z 830.746,A 0.000,B 0.000,C 90.000,E1 350.330} C_DIS
LIN {X -0.191,Y -461.199,Z 830.746,A 0.000,B 0.000,C 90.000,E1 350.274} C_DIS
LIN {X -0.092,Y -468.190,Z 830.743,A 0.000,B 0.000,C 90.000,E1 349.746} C_DIS
LIN {X -0.068,Y -483.447,Z 830.738,A 0.000,B 0.000,C 90.000,E1 348.814} C_DIS
LIN {X -0.120,Y -494.766,Z 830.734,A 0.000,B 0.000,C 90.000,E1 348.117} C_DIS
LIN {X -0.047,Y -509.102,Z 830.729,A 0.000,B 0.000,C 90.000,E1 347.173} C_DIS
LIN {X 0.095,Y -518.343,Z 830.725,A 0.000,B 0.000,C 90.000,E1 346.520} C_DIS
LIN {X 0.071,Y -530.643,Z 830.720,A 0.000,B 0.000,C 90.000,E1 345.644} C_DIS
LIN {X -0.079,Y -538.103,Z 830.717,A 0.000,B 0.000,C 90.000,E1 345.102} C_DIS
LIN {X -0.032,Y -545.304,Z 830.714,A 0.000,B 0.000,C 90.000,E1 344.519} C_DIS
LIN {X 0.057,Y -550.985,Z 830.711,A 0.000,B 0.000,C 90.000,E1 344.031} C_DIS
LIN {X 0.188,Y -559.209,Z 830.707,A 0.000,B 0.000,C 90.000,E1 343.268} C_DIS
LIN {X -0.024,Y -564.483,Z 830.704,A 0.000,B 0.000,C 90.000,E1 342.779} C_DIS
LIN {X 0.140,Y -569.550,Z 830.701,A 0.000,B 0.000,C 90.000,E1 342.236} C_DIS
LIN {X 0.141,Y -574.423,Z 830.698,A 0.000,B 0.000,C 90.000,E1 341.692} C_DIS
LIN {X -0.129,Y -580.256,Z 830.695,A 0.000,B 0.000,C 90.000,E1 341.040} C_DIS
LIN {X -0.169,Y -585.481,Z 830.691,A 0.000,B 0.000,C 90.000,E1 340.369} C_DIS
LIN {X -0.222,Y -591.252,Z 830.686,A 0.000,B 0.000,C 90.000,E1 339.571} C_DIS
LIN {X 0.291,Y -597.375,Z 830.681,A 0.000,B 0.000,C 90.000,E1 338.592} C_DIS
LIN {X -0.194,Y -602.261,Z 830.677,A 0.000,B 0.000,C 90.000,E1 337.847} C_DIS
LIN {X -0.186,Y -609.798,Z 830.670,A 0.000,B 0.000,C 90.000,E1 336.538} C_DIS
LIN {X -0.013,Y -614.938,Z 830.665,A 0.000,B 0.000,C 90.000,E1 335.613} C_DIS
LIN {X -0.091,Y -620.438,Z 830.659,A 0.000,B 0.000,C 90.000,E1 334.588} C_DIS
LIN {X -0.096,Y -624.321,Z 830.655,A 0.000,B 0.000,C 90.000,E1 333.819} C_DIS
LIN {X -0.039,Y -629.202,Z 830.649,A 0.000,B 0.000,C 90.000,E1 332.794} C_DIS
LIN {X 0.071,Y -633.723,Z 830.643,A 0.000,B 0.000,C 90.000,E1 331.769} C_DIS
LIN {X 0.036,Y -639.164,Z 830.636,A 0.000,B 0.000,C 90.000,E1 330.511} C_DIS
LIN {X -0.231,Y -644.289,Z 830.629,A 0.000,B 0.000,C 90.000,E1 329.282} C_DIS
LIN {X -0.250,Y -647.154,Z 830.625,A 0.000,B 0.000,C 90.000,E1 328.535} C_DIS
LIN {X -0.196,Y -652.298,Z 830.617,A 0.000,B 0.000,C 90.000,E1 327.041} C_DIS
LIN {X 0.320,Y -655.447,Z 830.611,A 0.000,B 0.000,C 90.000,E1 326.008} C_DIS
LIN {X -0.127,Y -657.736,Z 830.607,A 0.000,B 0.000,C 90.000,E1 325.308} C_DIS
LIN {X 0.015,Y -661.058,Z 830.600,A 0.000,B 0.000,C 90.000,E1 324.069} C_DIS
LIN {X 0.099,Y -663.464,Z 830.595,A 0.000,B 0.000,C 90.000,E1 323.084} C_DIS
LIN {X 0.117,Y -665.189,Z 830.591,A 0.000,B 0.000,C 90.000,E1 322.351} C_DIS
LIN {X 0.138,Y -667.222,Z 830.586,A 0.000,B 0.000,C 90.000,E1 321.376} C_DIS
LIN {X -0.236,Y -669.534,Z 830.579,A 0.000,B 0.000,C 90.000,E1 320.194} C_DIS
LIN {X 0.366,Y -671.638,Z 830.572,A 0.000,B 0.000,C 90.000,E1 318.933} C_DIS
LIN {X 0.011,Y -674.020,Z 830.564,A 0.000,B 0.000,C 90.000,E1 317.514} C_DIS
LIN {X 0.117,Y -675.124,Z 830.560,A 0.000,B 0.000,C 90.000,E1 316.782} C_DIS
LIN {X 0.363,Y -677.628,Z 830.549,A 0.000,B 0.000,C 90.000,E1 314.838} C_DIS
LIN {X 0.082,Y -678.936,Z 830.543,A 0.000,B 0.000,C 90.000,E1 313.662} C_DIS
LIN {X -0.128,Y -680.588,Z 830.535,A 0.000,B 0.000,C 90.000,E1 312.243} C_DIS
LIN {X -0.366,Y -681.854,Z 830.528,A 0.000,B 0.000,C 90.000,E1 311.067} C_DIS
LIN {X -0.081,Y -683.033,Z 830.521,A 0.000,B 0.000,C 90.000,E1 309.850} C_DIS
LIN {X 0.356,Y -684.314,Z 830.513,A 0.000,B 0.000,C 90.000,E1 308.382} C_DIS
LIN {X -0.144,Y -685.570,Z 830.505,A 0.000,B 0.000,C 90.000,E1 306.996} C_DIS
LIN {X -0.083,Y -686.775,Z 830.498,A 0.000,B 0.000,C 90.000,E1 305.564} C_DIS
LIN {X 0.165,Y -687.828,Z 830.490,A 0.000,B 0.000,C 90.000,E1 304.119} C_DIS
LIN {X 0.067,Y -688.812,Z 830.482,A 0.000,B 0.000,C 90.000,E1 302.704} C_DIS
LIN {X 0.360,Y -689.815,Z 830.474,A 0.000,B 0.000,C 90.000,E1 301.258} C_DIS
LIN {X -0.282,Y -690.727,Z 830.467,A 0.000,B 0.000,C 90.000,E1 300.129} C_DIS
LIN {X 0.169,Y -691.967,Z 830.458,A 0.000,B 0.000,C 90.000,E1 298.437} C_DIS
LIN {X -0.031,Y -693.422,Z 830.448,A 0.000,B 0.000,C 90.000,E1 296.565} C_DIS
LIN {X 0.342,Y -694.207,Z 830.442,A 0.000,B 0.000,C 90.000,E1 295.591} C_DIS
LIN {X -0.251,Y -695.227,Z 830.436,A 0.000,B 0.000,C 90.000,E1 294.463} C_DIS
LIN {X -0.414,Y -695.407,Z 830.432,A 0.000,B 0.000,C 90.000,E1 293.770} C_DIS
LIN {X 0.088,Y -694.655,Z 830.429,A 0.000,B 0.000,C 90.000,E1 293.259} C_DIS
LIN {X 0.062,Y -694.133,Z 830.428,A 0.000,B 0.000,C 90.000,E1 293.025} C_DIS
LIN {X 0.186,Y -693.564,Z 830.427,A 0.000,B 0.000,C 90.000,E1 292.898} C_DIS
LIN {X -0.237,Y -690.496,Z 830.425,A 0.000,B 0.000,C 90.000,E1 292.461} C_DIS
LIN {X -0.119,Y -689.554,Z 830.424,A 0.000,B 0.000,C 90.000,E1 292.333} C_DIS
LIN {X -0.006,Y -688.146,Z 830.423,A 0.000,B 0.000,C 90.000,E1 292.206} C_DIS
LIN {X -0.352,Y -684.553,Z 830.422,A 0.000,B 0.000,C 90.000,E1 292.025} C_DIS
LIN {X -0.290,Y -681.328,Z 830.421,A 0.000,B 0.000,C 90.000,E1 291.844} C_DIS
LIN {X 0.226,Y -679.332,Z 830.421,A 0.000,B 0.000,C 90.000,E1 291.716} C_DIS
LIN {X 0.158,Y -670.954,Z 830.419,A 0.000,B 0.000,C 90.000,E1 291.482} C_DIS
LIN {X -0.106,Y -662.017,Z 830.419,A 0.000,B 0.000,C 90.000,E1 291.334} C_DIS
LIN {X -0.001,Y -651.666,Z 830.418,A 0.000,B 0.000,C 90.000,E1 291.153} C_DIS
LIN {X -0.222,Y -641.965,Z 830.416,A 0.000,B 0.000,C 90.000,E1 290.972} C_DIS
LIN {X 0.116,Y -638.672,Z 830.416,A 0.000,B 0.000,C 90.000,E1 290.865} C_DIS
LIN {X -0.384,Y -632.277,Z 830.415,A 0.000,B 0.000,C 90.000,E1 290.737} C_DIS
LIN {X -0.021,Y -629.553,Z 830.415,A 0.000,B 0.000,C 90.000,E1 290.610} C_DIS
LIN {X 0.016,Y -624.142,Z 830.413,A 0.000,B 0.000,C 90.000,E1 290.375} C_DIS
LIN {X -0.293,Y -621.598,Z 830.412,A 0.000,B 0.000,C 90.000,E1 290.248} C_DIS
LIN {X -0.057,Y -620.032,Z 830.412,A 0.000,B 0.000,C 90.000,E1 290.120} C_DIS
LIN {X -0.091,Y -619.987,Z 830.412,A 0.000,B 0.000,C 90.000,E1 290.120} C_DIS
LIN {X -0.061,Y -619.047,Z 830.411,A 0.000,B 0.000,C 90.000,E1 289.939} C_DIS
LIN {X -0.105,Y -619.038,Z 830.411,A 0.000,B 0.000,C 90.000,E1 289.939} C_DIS
LIN {X 0.060,Y -619.519,Z 830.409,A 0.000,B 0.000,C 90.000,E1 289.631} C_DIS
LIN {X -0.240,Y -622.429,Z 830.406,A 0.000,B 0.000,C 90.000,E1 289.033} C_DIS
LIN {X -0.216,Y -626.801,Z 830.402,A 0.000,B 0.000,C 90.000,E1 288.308} C_DIS
LIN {X 0.157,Y -630.115,Z 830.398,A 0.000,B 0.000,C 90.000,E1 287.638} C_DIS
LIN {X -0.239,Y -633.089,Z 830.395,A 0.000,B 0.000,C 90.000,E1 287.040} C_DIS
LIN {X -0.007,Y -636.169,Z 830.390,A 0.000,B 0.000,C 90.000,E1 286.260} C_DIS
LIN {X 0.256,Y -638.628,Z 830.386,A 0.000,B 0.000,C 90.000,E1 285.481} C_DIS
LIN {X -0.081,Y -640.079,Z 830.383,A 0.000,B 0.000,C 90.000,E1 285.009} C_DIS
LIN {X 0.055,Y -641.732,Z 830.379,A 0.000,B 0.000,C 90.000,E1 284.245} C_DIS
LIN {X -0.258,Y -642.664,Z 830.376,A 0.000,B 0.000,C 90.000,E1 283.772} C_DIS
LIN {X -0.091,Y -643.395,Z 830.372,A 0.000,B 0.000,C 90.000,E1 283.008} C_DIS
LIN {X 0.236,Y -643.582,Z 830.370,A 0.000,B 0.000,C 90.000,E1 282.479} C_DIS
LIN {X -0.067,Y -643.465,Z 830.367,A 0.000,B 0.000,C 90.000,E1 282.007} C_DIS
LIN {X 0.104,Y -642.900,Z 830.363,A 0.000,B 0.000,C 90.000,E1 281.243} C_DIS
LIN {X -0.329,Y -642.123,Z 830.360,A 0.000,B 0.000,C 90.000,E1 280.782} C_DIS
LIN {X -0.016,Y -641.067,Z 830.357,A 0.000,B 0.000,C 90.000,E1 280.254} C_DIS
LIN {X 0.287,Y -639.759,Z 830.354,A 0.000,B 0.000,C 90.000,E1 279.726} C_DIS
LIN {X 0.012,Y -638.968,Z 830.353,A 0.000,B 0.000,C 90.000,E1 279.500} C_DIS
LIN {X 0.298,Y -637.024,Z 830.350,A 0.000,B 0.000,C 90.000,E1 278.973} C_DIS
LIN {X -0.159,Y -634.617,Z 830.347,A 0.000,B 0.000,C 90.000,E1 278.511} C_DIS
LIN {X -0.002,Y -631.865,Z 830.344,A 0.000,B 0.000,C 90.000,E1 277.992} C_DIS
LIN {X 0.136,Y -628.603,Z 830.342,A 0.000,B 0.000,C 90.000,E1 277.473} C_DIS
LIN {X 0.178,Y -623.637,Z 830.338,A 0.000,B 0.000,C 90.000,E1 276.834} C_DIS
LIN {X -0.202,Y -620.001,Z 830.336,A 0.000,B 0.000,C 90.000,E1 276.486} C_DIS
LIN {X 0.283,Y -618.737,Z 830.335,A 0.000,B 0.000,C 90.000,E1 276.315} C_DIS
LIN {X 0.225,Y -613.139,Z 830.333,A 0.000,B 0.000,C 90.000,E1 275.853} C_DIS
LIN {X 0.263,Y -611.619,Z 830.332,A 0.000,B 0.000,C 90.000,E1 275.739} C_DIS
LIN {X 0.054,Y -606.620,Z 830.330,A 0.000,B 0.000,C 90.000,E1 275.454} C_DIS
LIN {X 0.285,Y -601.612,Z 830.329,A 0.000,B 0.000,C 90.000,E1 275.163} C_DIS
LIN {X -0.236,Y -592.948,Z 830.327,A 0.000,B 0.000,C 90.000,E1 274.816} C_DIS
LIN {X -0.242,Y -585.873,Z 830.325,A 0.000,B 0.000,C 90.000,E1 274.531} C_DIS
LIN {X 0.259,Y -578.599,Z 830.324,A 0.000,B 0.000,C 90.000,E1 274.245} C_DIS
LIN {X -0.004,Y -572.521,Z 830.323,A 0.000,B 0.000,C 90.000,E1 274.131} C_DIS
LIN {X -0.214,Y -565.453,Z 830.323,A 0.000,B 0.000,C 90.000,E1 274.069} C_DIS
LIN {X 0.180,Y -558.707,Z 830.322,A 0.000,B 0.000,C 90.000,E1 274.012} C_DIS
LIN {X 0.123,Y -553.565,Z 830.322,A 0.000,B 0.000,C 90.000,E1 274.012} C_DIS
LIN {X -0.036,Y -550.505,Z 830.322,A 0.000,B 0.000,C 90.000,E1 273.955} C_DIS
LIN {X -0.091,Y -550.308,Z 830.322,A 0.000,B 0.000,C 90.000,E1 273.955} C_DIS
LIN {X -0.117,Y -549.737,Z 830.321,A 0.000,B 0.000,C 90.000,E1 273.784} C_DIS
LIN {X 0.233,Y -548.972,Z 830.319,A 0.000,B 0.000,C 90.000,E1 273.326} C_DIS
LIN {X -0.261,Y -546.000,Z 830.300,A 0.000,B 0.000,C 90.000,E1 270.000} C_DIS
LIN {X -0.060,Y -544.965,Z 830.292,A 0.000,B 0.000,C 90.000,E1 268.568} C_DIS
LIN {X 0.066,Y -544.410,Z 830.287,A 0.000,B 0.000,C 90.000,E1 267.707} C_DIS
LIN {X -0.265,Y -543.290,Z 830.278,A 0.000,B 0.000,C 90.000,E1 266.045} C_DIS
LIN {X 0.008,Y -541.980,Z 830.267,A 0.000,B 0.000,C 90.000,E1 264.033} C_DIS
LIN {X 0.230,Y -540.882,Z 830.259,A 0.000,B 0.000,C 90.000,E1 262.591} C_DIS
LIN {X 0.094,Y -538.717,Z 830.246,A 0.000,B 0.000,C 90.000,E1 260.330} C_DIS
LIN {X -0.036,Y -537.055,Z 830.237,A 0.000,B 0.000,C 90.000,E1 258.634} C_DIS
LIN {X -0.141,Y -535.035,Z 830.226,A 0.000,B 0.000,C 90.000,E1 256.645} C_DIS
LIN {X -0.053,Y -532.769,Z 830.215,A 0.000,B 0.000,C 90.000,E1 254.629} C_DIS
LIN {X -0.062,Y -530.810,Z 830.205,A 0.000,B 0.000,C 90.000,E1 252.906} C_DIS
LIN {X 0.201,Y -528.662,Z 830.195,A 0.000,B 0.000,C 90.000,E1 251.148} C_DIS
LIN {X 0.243,Y -526.766,Z 830.187,A 0.000,B 0.000,C 90.000,E1 249.699} C_DIS
LIN {X 0.102,Y -524.301,Z 830.178,A 0.000,B 0.000,C 90.000,E1 247.975} C_DIS
LIN {X -0.048,Y -522.190,Z 830.170,A 0.000,B 0.000,C 90.000,E1 246.538} C_DIS
LIN {X -0.091,Y -519.451,Z 830.160,A 0.000,B 0.000,C 90.000,E1 244.793} C_DIS
LIN {X -0.249,Y -517.563,Z 830.153,A 0.000,B 0.000,C 90.000,E1 243.640} C_DIS
LIN {X 0.038,Y -514.441,Z 830.144,A 0.000,B 0.000,C 90.000,E1 241.847} C_DIS
LIN {X -0.054,Y -511.848,Z 830.135,A 0.000,B 0.000,C 90.000,E1 240.383} C_DIS
LIN {X -0.111,Y -508.542,Z 830.126,A 0.000,B 0.000,C 90.000,E1 238.614} C_DIS
LIN {X 0.063,Y -506.190,Z 830.119,A 0.000,B 0.000,C 90.000,E1 237.406} C_DIS
LIN {X -0.058,Y -503.056,Z 830.111,A 0.000,B 0.000,C 90.000,E1 235.928} C_DIS
LIN {X 0.017,Y -501.054,Z 830.106,A 0.000,B 0.000,C 90.000,E1 235.022} C_DIS
LIN {X 0.217,Y -497.597,Z 830.097,A 0.000,B 0.000,C 90.000,E1 233.497} C_DIS
LIN {X 0.097,Y -493.307,Z 830.087,A 0.000,B 0.000,C 90.000,E1 231.698} C_DIS
LIN {X -0.206,Y -487.552,Z 830.074,A 0.000,B 0.000,C 90.000,E1 229.299} C_DIS
LIN {X -0.259,Y -484.696,Z 830.067,A 0.000,B 0.000,C 90.000,E1 228.081} C_DIS
LIN {X -0.228,Y -481.233,Z 830.058,A 0.000,B 0.000,C 90.000,E1 226.539} C_DIS
LIN {X 0.156,Y -479.137,Z 830.053,A 0.000,B 0.000,C 90.000,E1 225.567} C_DIS
LIN {X 0.065,Y -475.856,Z 830.045,A 0.000,B 0.000,C 90.000,E1 224.028} C_DIS
LIN {X 0.115,Y -471.210,Z 830.033,A 0.000,B 0.000,C 90.000,E1 221.838} C_DIS
LIN {X 0.078,Y -466.503,Z 830.020,A 0.000,B 0.000,C 90.000,E1 219.644} C_DIS
LIN {X -0.024,Y -461.916,Z 830.008,A 0.000,B 0.000,C 90.000,E1 217.443} C_DIS
LIN {X -0.009,Y -458.640,Z 829.999,A 0.000,B 0.000,C 90.000,E1 215.851} C_DIS
LIN {X 0.053,Y -456.026,Z 829.992,A 0.000,B 0.000,C 90.000,E1 214.565} C_DIS
LIN {X 0.151,Y -451.838,Z 829.981,A 0.000,B 0.000,C 90.000,E1 212.625} C_DIS
LIN {X -0.101,Y -447.812,Z 829.971,A 0.000,B 0.000,C 90.000,E1 210.718} C_DIS
LIN {X -0.069,Y -443.220,Z 829.958,A 0.000,B 0.000,C 90.000,E1 208.437} C_DIS
LIN {X -0.034,Y -440.046,Z 829.949,A 0.000,B 0.000,C 90.000,E1 206.796} C_DIS
LIN {X -0.069,Y -436.742,Z 829.940,A 0.000,B 0.000,C 90.000,E1 205.155} C_DIS
LIN {X 0.059,Y -432.645,Z 829.929,A 0.000,B 0.000,C 90.000,E1 203.153} C_DIS
LIN {X -0.111,Y -428.140,Z 829.916,A 0.000,B 0.000,C 90.000,E1 200.844} C_DIS
LIN {X -0.104,Y -425.580,Z 829.908,A 0.000,B 0.000,C 90.000,E1 199.504} C_DIS
LIN {X 0.093,Y -421.564,Z 829.897,A 0.000,B 0.000,C 90.000,E1 197.457} C_DIS
LIN {X -0.138,Y -419.034,Z 829.890,A 0.000,B 0.000,C 90.000,E1 196.134} C_DIS
LIN {X 0.071,Y -415.170,Z 829.878,A 0.000,B 0.000,C 90.000,E1 194.064} C_DIS
LIN {X 0.092,Y -411.106,Z 829.867,A 0.000,B 0.000,C 90.000,E1 192.007} C_DIS
LIN {X -0.070,Y -407.175,Z 829.855,A 0.000,B 0.000,C 90.000,E1 189.962} C_DIS
LIN {X -0.003,Y -403.265,Z 829.844,A 0.000,B 0.000,C 90.000,E1 187.871} C_DIS
LIN {X -0.126,Y -399.977,Z 829.834,A 0.000,B 0.000,C 90.000,E1 186.144} C_DIS
LIN {X -0.076,Y -395.057,Z 829.818,A 0.000,B 0.000,C 90.000,E1 183.326} C_DIS
LIN {X 0.002,Y -390.083,Z 829.799,A 0.000,B 0.000,C 90.000,E1 179.771} C_DIS
LIN {X 0.045,Y -388.301,Z 829.791,A 0.000,B 0.000,C 90.000,E1 178.339} C_DIS
LIN {X -0.014,Y -386.078,Z 829.781,A 0.000,B 0.000,C 90.000,E1 176.560} C_DIS
LIN {X 0.186,Y -383.444,Z 829.769,A 0.000,B 0.000,C 90.000,E1 174.375} C_DIS
LIN {X 0.173,Y -380.163,Z 829.753,A 0.000,B 0.000,C 90.000,E1 171.489} C_DIS
LIN {X 0.082,Y -378.438,Z 829.743,A 0.000,B 0.000,C 90.000,E1 169.690} C_DIS
LIN {X 0.125,Y -377.111,Z 829.735,A 0.000,B 0.000,C 90.000,E1 168.229} C_DIS
LIN {X 0.005,Y -373.733,Z 829.710,A 0.000,B 0.000,C 90.000,E1 163.866} C_DIS
LIN {X 0.163,Y -372.651,Z 829.696,A 0.000,B 0.000,C 90.000,E1 161.275} C_DIS
LIN {X 0.103,Y -372.657,Z 829.684,A 0.000,B 0.000,C 90.000,E1 159.082} C_DIS
LIN {X 0.211,Y -373.487,Z 829.674,A 0.000,B 0.000,C 90.000,E1 157.230} C_DIS
LIN {X -0.090,Y -374.472,Z 829.668,A 0.000,B 0.000,C 90.000,E1 156.177} C_DIS
LIN {X 0.110,Y -376.070,Z 829.661,A 0.000,B 0.000,C 90.000,E1 155.049} C_DIS
LIN {X -0.107,Y -376.852,Z 829.659,A 0.000,B 0.000,C 90.000,E1 154.717} C_DIS
LIN {X 0.022,Y -377.487,Z 829.657,A 0.000,B 0.000,C 90.000,E1 154.332} C_DIS
LIN {X -0.011,Y -378.475,Z 829.655,A 0.000,B 0.000,C 90.000,E1 153.973} C_DIS
LIN {X -0.028,Y -379.747,Z 829.652,A 0.000,B 0.000,C 90.000,E1 153.435} C_DIS
LIN {X 0.088,Y -382.046,Z 829.648,A 0.000,B 0.000,C 90.000,E1 152.692} C_DIS
LIN {X 0.065,Y -384.289,Z 829.645,A 0.000,B 0.000,C 90.000,E1 152.153} C_DIS
LIN {X 0.056,Y -384.850,Z 829.644,A 0.000,B 0.000,C 90.000,E1 151.975} C_DIS
LIN {X 0.016,Y -387.707,Z 829.641,A 0.000,B 0.000,C 90.000,E1 151.435} C_DIS
LIN {X -0.152,Y -391.870,Z 829.638,A 0.000,B 0.000,C 90.000,E1 150.923} C_DIS
LIN {X 0.010,Y -396.478,Z 829.635,A 0.000,B 0.000,C 90.000,E1 150.383} C_DIS
LIN {X 0.131,Y -398.221,Z 829.635,A 0.000,B 0.000,C 90.000,E1 150.205} C_DIS
LIN {X 0.254,Y -405.950,Z 829.632,A 0.000,B 0.000,C 90.000,E1 149.665} C_DIS
LIN {X 0.157,Y -425.153,Z 829.627,A 0.000,B 0.000,C 90.000,E1 148.742} C_DIS
LIN {X -0.041,Y -431.806,Z 829.625,A 0.000,B 0.000,C 90.000,E1 148.408} C_DIS
LIN {X 0.243,Y -437.953,Z 829.622,A 0.000,B 0.000,C 90.000,E1 147.995} C_DIS
LIN {X 0.130,Y -444.403,Z 829.620,A 0.000,B 0.000,C 90.000,E1 147.582} C_DIS
LIN {X 0.171,Y -450.338,Z 829.617,A 0.000,B 0.000,C 90.000,E1 147.120} C_DIS
LIN {X 0.236,Y -456.122,Z 829.615,A 0.000,B 0.000,C 90.000,E1 146.628} C_DIS
LIN {X -0.184,Y -463.221,Z 829.611,A 0.000,B 0.000,C 90.000,E1 146.008} C_DIS
LIN {X 0.058,Y -465.989,Z 829.610,A 0.000,B 0.000,C 90.000,E1 145.722} C_DIS
LIN {X -0.025,Y -472.719,Z 829.606,A 0.000,B 0.000,C 90.000,E1 145.022} C_DIS
LIN {X 0.078,Y -482.819,Z 829.599,A 0.000,B 0.000,C 90.000,E1 143.783} C_DIS
LIN {X -0.110,Y -485.339,Z 829.597,A 0.000,B 0.000,C 90.000,E1 143.497} C_DIS
LIN {X 0.222,Y -489.789,Z 829.594,A 0.000,B 0.000,C 90.000,E1 142.844} C_DIS
LIN {X -0.246,Y -496.173,Z 829.589,A 0.000,B 0.000,C 90.000,E1 141.984} C_DIS
LIN {X 0.244,Y -504.132,Z 829.582,A 0.000,B 0.000,C 90.000,E1 140.723} C_DIS
LIN {X 0.132,Y -508.717,Z 829.578,A 0.000,B 0.000,C 90.000,E1 139.989} C_DIS
LIN {X -0.083,Y -514.732,Z 829.572,A 0.000,B 0.000,C 90.000,E1 138.976} C_DIS
LIN {X -0.106,Y -518.873,Z 829.568,A 0.000,B 0.000,C 90.000,E1 138.243} C_DIS
LIN {X -0.095,Y -526.508,Z 829.560,A 0.000,B 0.000,C 90.000,E1 136.782} C_DIS
LIN {X 0.281,Y -531.744,Z 829.554,A 0.000,B 0.000,C 90.000,E1 135.729} C_DIS
LIN {X 0.125,Y -540.520,Z 829.545,A 0.000,B 0.000,C 90.000,E1 134.028} C_DIS
LIN {X -0.255,Y -545.966,Z 829.538,A 0.000,B 0.000,C 90.000,E1 132.933} C_DIS
LIN {X -0.152,Y -552.184,Z 829.531,A 0.000,B 0.000,C 90.000,E1 131.515} C_DIS
LIN {X 0.032,Y -556.834,Z 829.524,A 0.000,B 0.000,C 90.000,E1 130.378} C_DIS
LIN {X -0.166,Y -560.081,Z 829.520,A 0.000,B 0.000,C 90.000,E1 129.564} C_DIS
LIN {X 0.110,Y -563.132,Z 829.515,A 0.000,B 0.000,C 90.000,E1 128.705} C_DIS
LIN {X 0.094,Y -566.734,Z 829.509,A 0.000,B 0.000,C 90.000,E1 127.604} C_DIS
LIN {X -0.002,Y -569.319,Z 829.504,A 0.000,B 0.000,C 90.000,E1 126.790} C_DIS
LIN {X 0.249,Y -570.782,Z 829.501,A 0.000,B 0.000,C 90.000,E1 126.217} C_DIS
LIN {X 0.178,Y -572.004,Z 829.498,A 0.000,B 0.000,C 90.000,E1 125.678} C_DIS
LIN {X -0.067,Y -573.904,Z 829.492,A 0.000,B 0.000,C 90.000,E1 124.612} C_DIS
LIN {X 0.181,Y -575.622,Z 829.486,A 0.000,B 0.000,C 90.000,E1 123.499} C_DIS
LIN {X 0.155,Y -576.269,Z 829.483,A 0.000,B 0.000,C 90.000,E1 122.959} C_DIS
LIN {X 0.282,Y -577.052,Z 829.479,A 0.000,B 0.000,C 90.000,E1 122.133} C_DIS
LIN {X 0.268,Y -577.482,Z 829.476,A 0.000,B 0.000,C 90.000,E1 121.592} C_DIS
LIN {X 0.101,Y -577.679,Z 829.471,A 0.000,B 0.000,C 90.000,E1 120.797} C_DIS
LIN {X -0.211,Y -577.598,Z 829.465,A 0.000,B 0.000,C 90.000,E1 119.745} C_DIS
LIN {X -0.224,Y -577.363,Z 829.462,A 0.000,B 0.000,C 90.000,E1 119.205} C_DIS
LIN {X 0.113,Y -576.840,Z 829.458,A 0.000,B 0.000,C 90.000,E1 118.359} C_DIS
LIN {X 0.142,Y -575.427,Z 829.450,A 0.000,B 0.000,C 90.000,E1 117.001} C_DIS
LIN {X -0.163,Y -574.619,Z 829.447,A 0.000,B 0.000,C 90.000,E1 116.488} C_DIS
LIN {X -0.112,Y -572.903,Z 829.443,A 0.000,B 0.000,C 90.000,E1 115.668} C_DIS
LIN {X 0.087,Y -571.244,Z 829.440,A 0.000,B 0.000,C 90.000,E1 115.103} C_DIS
LIN {X -0.243,Y -569.251,Z 829.437,A 0.000,B 0.000,C 90.000,E1 114.591} C_DIS
LIN {X -0.158,Y -566.171,Z 829.433,A 0.000,B 0.000,C 90.000,E1 113.898} C_DIS
LIN {X -0.248,Y -565.423,Z 829.432,A 0.000,B 0.000,C 90.000,E1 113.770} C_DIS
LIN {X -0.103,Y -563.232,Z 829.429,A 0.000,B 0.000,C 90.000,E1 113.206} C_DIS
LIN {X -0.141,Y -562.695,Z 829.428,A 0.000,B 0.000,C 90.000,E1 113.003} C_DIS
LIN {X 0.210,Y -562.760,Z 829.427,A 0.000,B 0.000,C 90.000,E1 112.823} C_DIS
LIN {X 0.114,Y -562.531,Z 829.424,A 0.000,B 0.000,C 90.000,E1 112.280} C_DIS
LIN {X 0.064,Y -562.630,Z 829.423,A 0.000,B 0.000,C 90.000,E1 112.099} C_DIS
LIN {X 0.183,Y -562.581,Z 829.420,A 0.000,B 0.000,C 90.000,E1 111.535} C_DIS
LIN {X -0.022,Y -562.695,Z 829.418,A 0.000,B 0.000,C 90.000,E1 111.280} C_DIS
LIN {X -0.086,Y -562.586,Z 829.409,A 0.000,B 0.000,C 90.000,E1 109.631} C_DIS
LIN {X -0.116,Y -562.328,Z 829.395,A 0.000,B 0.000,C 90.000,E1 107.149} C_DIS
LIN {X -0.030,Y -563.159,Z 829.377,A 0.000,B 0.000,C 90.000,E1 103.828} C_DIS
LIN {X -0.221,Y -564.535,Z 829.363,A 0.000,B 0.000,C 90.000,E1 101.366} C_DIS
LIN {X -0.164,Y -565.995,Z 829.352,A 0.000,B 0.000,C 90.000,E1 99.434} C_DIS
LIN {X 0.117,Y -567.107,Z 829.343,A 0.000,B 0.000,C 90.000,E1 97.757} C_DIS
LIN {X -0.205,Y -568.074,Z 829.334,A 0.000,B 0.000,C 90.000,E1 96.144} C_DIS
LIN {X 0.236,Y -568.509,Z 829.330,A 0.000,B 0.000,C 90.000,E1 95.277} C_DIS
LIN {X -0.230,Y -569.145,Z 829.322,A 0.000,B 0.000,C 90.000,E1 93.955} C_DIS
LIN {X -0.153,Y -569.656,Z 829.314,A 0.000,B 0.000,C 90.000,E1 92.579} C_DIS
LIN {X 0.193,Y -570.276,Z 829.304,A 0.000,B 0.000,C 90.000,E1 90.630} C_DIS
LIN {X -0.158,Y -570.696,Z 829.295,A 0.000,B 0.000,C 90.000,E1 89.026} C_DIS
LIN {X -0.051,Y -571.044,Z 829.287,A 0.000,B 0.000,C 90.000,E1 87.650} C_DIS
LIN {X -0.212,Y -571.412,Z 829.276,A 0.000,B 0.000,C 90.000,E1 85.755} C_DIS
LIN {X 0.068,Y -571.666,Z 829.267,A 0.000,B 0.000,C 90.000,E1 84.090} C_DIS
LIN {X -0.283,Y -572.018,Z 829.260,A 0.000,B 0.000,C 90.000,E1 82.761} C_DIS
LIN {X 0.054,Y -572.616,Z 829.246,A 0.000,B 0.000,C 90.000,E1 80.274} C_DIS
LIN {X 0.112,Y -573.106,Z 829.237,A 0.000,B 0.000,C 90.000,E1 78.634} C_DIS
LIN {X -0.333,Y -573.403,Z 829.231,A 0.000,B 0.000,C 90.000,E1 77.589} C_DIS
LIN {X -0.129,Y -573.713,Z 829.222,A 0.000,B 0.000,C 90.000,E1 75.936} C_DIS
LIN {X -0.112,Y -573.889,Z 829.214,A 0.000,B 0.000,C 90.000,E1 74.574} C_DIS
LIN {X -0.112,Y -573.887,Z 829.204,A 0.000,B 0.000,C 90.000,E1 72.670} C_DIS
LIN {X -0.132,Y -573.758,Z 829.195,A 0.000,B 0.000,C 90.000,E1 71.040} C_DIS
LIN {X -0.134,Y -573.479,Z 829.184,A 0.000,B 0.000,C 90.000,E1 69.135} C_DIS
LIN {X 0.030,Y -573.122,Z 829.175,A 0.000,B 0.000,C 90.000,E1 67.486} C_DIS
LIN {X -0.138,Y -572.604,Z 829.166,A 0.000,B 0.000,C 90.000,E1 65.869} C_DIS
LIN {X -0.276,Y -572.195,Z 829.160,A 0.000,B 0.000,C 90.000,E1 64.793} C_DIS
LIN {X 0.015,Y -571.417,Z 829.151,A 0.000,B 0.000,C 90.000,E1 63.127} C_DIS
LIN {X -0.048,Y -570.628,Z 829.143,A 0.000,B 0.000,C 90.000,E1 61.769} C_DIS
LIN {X 0.216,Y -570.041,Z 829.139,A 0.000,B 0.000,C 90.000,E1 60.923} C_DIS
LIN {X -0.024,Y -569.275,Z 829.134,A 0.000,B 0.000,C 90.000,E1 60.127} C_DIS
LIN {X 0.329,Y -568.112,Z 829.128,A 0.000,B 0.000,C 90.000,E1 58.997} C_DIS
LIN {X -0.013,Y -566.403,Z 829.120,A 0.000,B 0.000,C 90.000,E1 57.661} C_DIS
LIN {X 0.118,Y -564.818,Z 829.114,A 0.000,B 0.000,C 90.000,E1 56.548} C_DIS
LIN {X -0.085,Y -563.004,Z 829.108,A 0.000,B 0.000,C 90.000,E1 55.468} C_DIS
LIN {X 0.222,Y -561.408,Z 829.104,A 0.000,B 0.000,C 90.000,E1 54.609} C_DIS
LIN {X -0.170,Y -558.980,Z 829.097,A 0.000,B 0.000,C 90.000,E1 53.543} C_DIS
LIN {X 0.101,Y -556.961,Z 829.093,A 0.000,B 0.000,C 90.000,E1 52.683} C_DIS
LIN {X 0.346,Y -554.673,Z 829.088,A 0.000,B 0.000,C 90.000,E1 51.823} C_DIS
LIN {X 0.061,Y -553.014,Z 829.085,A 0.000,B 0.000,C 90.000,E1 51.295} C_DIS
LIN {X 0.195,Y -551.247,Z 829.082,A 0.000,B 0.000,C 90.000,E1 50.723} C_DIS
LIN {X -0.056,Y -548.271,Z 829.077,A 0.000,B 0.000,C 90.000,E1 49.908} C_DIS
LIN {X 0.035,Y -546.169,Z 829.074,A 0.000,B 0.000,C 90.000,E1 49.337} C_DIS
LIN {X 0.273,Y -541.867,Z 829.069,A 0.000,B 0.000,C 90.000,E1 48.324} C_DIS
LIN {X -0.098,Y -539.189,Z 829.066,A 0.000,B 0.000,C 90.000,E1 47.796} C_DIS
LIN {X -0.125,Y -536.261,Z 829.062,A 0.000,B 0.000,C 90.000,E1 47.229} C_DIS
LIN {X 0.220,Y -533.048,Z 829.059,A 0.000,B 0.000,C 90.000,E1 46.620} C_DIS
LIN {X 0.351,Y -528.615,Z 829.055,A 0.000,B 0.000,C 90.000,E1 45.891} C_DIS
LIN {X 0.093,Y -525.769,Z 829.053,A 0.000,B 0.000,C 90.000,E1 45.486} C_DIS
LIN {X -0.023,Y -521.550,Z 829.050,A 0.000,B 0.000,C 90.000,E1 44.919} C_DIS
LIN {X -0.169,Y -516.989,Z 829.046,A 0.000,B 0.000,C 90.000,E1 44.352} C_DIS
LIN {X 0.248,Y -513.371,Z 829.044,A 0.000,B 0.000,C 90.000,E1 43.866} C_DIS
LIN {X 0.071,Y -508.586,Z 829.041,A 0.000,B 0.000,C 90.000,E1 43.338} C_DIS
LIN {X -0.057,Y -503.147,Z 829.038,A 0.000,B 0.000,C 90.000,E1 42.771} C_DIS
LIN {X 0.150,Y -494.813,Z 829.033,A 0.000,B 0.000,C 90.000,E1 41.919} C_DIS
LIN {X -0.041,Y -487.327,Z 829.029,A 0.000,B 0.000,C 90.000,E1 41.272} C_DIS
LIN {X -0.178,Y -481.154,Z 829.026,A 0.000,B 0.000,C 90.000,E1 40.782} C_DIS
LIN {X -0.206,Y -473.540,Z 829.023,A 0.000,B 0.000,C 90.000,E1 40.172} C_DIS
LIN {X -0.058,Y -464.004,Z 829.019,A 0.000,B 0.000,C 90.000,E1 39.439} C_DIS
LIN {X 0.125,Y -456.121,Z 829.016,A 0.000,B 0.000,C 90.000,E1 38.830} C_DIS
LIN {X -0.126,Y -441.807,Z 829.010,A 0.000,B 0.000,C 90.000,E1 37.810} C_DIS
LIN {X 0.139,Y -418.365,Z 829.000,A 0.000,B 0.000,C 90.000,E1 35.931} C_DIS
LIN {X -0.139,Y -406.302,Z 828.994,A 0.000,B 0.000,C 90.000,E1 34.898} C_DIS
LIN {X 0.030,Y -402.026,Z 828.991,A 0.000,B 0.000,C 90.000,E1 34.452} C_DIS
LIN {X 0.045,Y -396.919,Z 828.988,A 0.000,B 0.000,C 90.000,E1 33.833} C_DIS
LIN {X 0.190,Y -396.747,Z 828.988,A 0.000,B 0.000,C 90.000,E1 33.785} C_DIS
LIN {X 0.153,Y -396.736,Z 828.988,A 0.000,B 0.000,C 90.000,E1 33.785} C_DIS
LIN {X 0.139,Y -393.769,Z 828.977,A 0.000,B 0.000,C 90.000,E1 31.799} C_DIS
LIN {X 0.064,Y -391.711,Z 828.971,A 0.000,B 0.000,C 90.000,E1 30.747} C_DIS
LIN {X -0.135,Y -393.456,Z 828.951,A 0.000,B 0.000,C 90.000,E1 27.129} C_DIS
LIN {X 0.128,Y -395.352,Z 828.935,A 0.000,B 0.000,C 90.000,E1 24.259} C_DIS
LIN {X 0.118,Y -397.251,Z 828.921,A 0.000,B 0.000,C 90.000,E1 21.791} C_DIS
LIN {X 0.243,Y -399.769,Z 828.906,A 0.000,B 0.000,C 90.000,E1 18.960} C_DIS
LIN {X -0.049,Y -402.449,Z 828.892,A 0.000,B 0.000,C 90.000,E1 16.551} C_DIS
LIN {X -0.006,Y -406.775,Z 828.875,A 0.000,B 0.000,C 90.000,E1 13.411} C_DIS
LIN {X -0.075,Y -411.753,Z 828.857,A 0.000,B 0.000,C 90.000,E1 10.310} C_DIS
LIN {X 0.198,Y -415.959,Z 828.844,A 0.000,B 0.000,C 90.000,E1 7.871} C_DIS
LIN {X -0.068,Y -418.381,Z 828.836,A 0.000,B 0.000,C 90.000,E1 6.543} C_DIS
LIN {X 0.166,Y -422.099,Z 828.825,A 0.000,B 0.000,C 90.000,E1 4.473} C_DIS
LIN {X 0.172,Y -427.444,Z 828.810,A 0.000,B 0.000,C 90.000,E1 1.776} C_DIS
LIN {X -0.108,Y -433.213,Z 828.795,A 0.000,B 0.000,C 90.000,E1 359.141} C_DIS
LIN {X 0.020,Y -437.902,Z 828.784,A 0.000,B 0.000,C 90.000,E1 357.135} C_DIS
LIN {X -0.128,Y -442.728,Z 828.773,A 0.000,B 0.000,C 90.000,E1 355.179} C_DIS
LIN {X -0.158,Y -447.695,Z 828.762,A 0.000,B 0.000,C 90.000,E1 353.223} C_DIS
LIN {X 0.084,Y -451.237,Z 828.755,A 0.000,B 0.000,C 90.000,E1 351.894} C_DIS
LIN {X 0.036,Y -453.578,Z 828.751,A 0.000,B 0.000,C 90.000,E1 351.254} C_DIS
LIN {X -0.058,Y -455.488,Z 828.749,A 0.000,B 0.000,C 90.000,E1 350.849} C_DIS
LIN {X -0.070,Y -459.513,Z 828.746,A 0.000,B 0.000,C 90.000,E1 350.330} C_DIS
LIN {X 0.083,Y -460.992,Z 828.745,A 0.000,B 0.000,C 90.000,E1 350.151} C_DIS
LIN {X -0.141,Y -467.911,Z 828.742,A 0.000,B 0.000,C 90.000,E1 349.634} C_DIS
LIN {X 0.126,Y -483.471,Z 828.737,A 0.000,B 0.000,C 90.000,E1 348.634} C_DIS
LIN {X 0.128,Y -490.068,Z 828.735,A 0.000,B 0.000,C 90.000,E1 348.229} C_DIS
LIN {X -0.093,Y -505.936,Z 828.729,A 0.000,B 0.000,C 90.000,E1 347.229} C_DIS
LIN {X -0.020,Y -515.285,Z 828.726,A 0.000,B 0.000,C 90.000,E1 346.589} C_DIS
LIN {X 0.164,Y -527.597,Z 828.721,A 0.000,B 0.000,C 90.000,E1 345.700} C_DIS
LIN {X -0.075,Y -535.160,Z 828.718,A 0.000,B 0.000,C 90.000,E1 345.172} C_DIS
LIN {X 0.159,Y -542.491,Z 828.714,A 0.000,B 0.000,C 90.000,E1 344.574} C_DIS
LIN {X 0.237,Y -549.688,Z 828.711,A 0.000,B 0.000,C 90.000,E1 343.976} C_DIS
LIN {X -0.026,Y -557.878,Z 828.707,A 0.000,B 0.000,C 90.000,E1 343.268} C_DIS
LIN {X -0.188,Y -563.218,Z 828.704,A 0.000,B 0.000,C 90.000,E1 342.779} C_DIS
LIN {X 0.061,Y -568.274,Z 828.701,A 0.000,B 0.000,C 90.000,E1 342.236} C_DIS
LIN {X 0.144,Y -573.215,Z 828.698,A 0.000,B 0.000,C 90.000,E1 341.692} C_DIS
LIN {X -0.085,Y -579.106,Z 828.695,A 0.000,B 0.000,C 90.000,E1 341.040} C_DIS
LIN {X -0.207,Y -585.479,Z 828.690,A 0.000,B 0.000,C 90.000,E1 340.242} C_DIS
LIN {X 0.293,Y -591.243,Z 828.686,A 0.000,B 0.000,C 90.000,E1 339.390} C_DIS
LIN {X -0.199,Y -595.634,Z 828.682,A 0.000,B 0.000,C 90.000,E1 338.773} C_DIS
LIN {X -0.148,Y -600.632,Z 828.678,A 0.000,B 0.000,C 90.000,E1 337.975} C_DIS
LIN {X -0.047,Y -605.264,Z 828.673,A 0.000,B 0.000,C 90.000,E1 337.177} C_DIS
LIN {X 0.295,Y -611.281,Z 828.667,A 0.000,B 0.000,C 90.000,E1 336.102} C_DIS
LIN {X -0.074,Y -616.361,Z 828.662,A 0.000,B 0.000,C 90.000,E1 335.229} C_DIS
LIN {X -0.126,Y -621.146,Z 828.657,A 0.000,B 0.000,C 90.000,E1 334.332} C_DIS
LIN {X -0.122,Y -624.992,Z 828.653,A 0.000,B 0.000,C 90.000,E1 333.563} C_DIS
LIN {X -0.069,Y -629.267,Z 828.648,A 0.000,B 0.000,C 90.000,E1 332.666} C_DIS
LIN {X 0.040,Y -633.784,Z 828.643,A 0.000,B 0.000,C 90.000,E1 331.641} C_DIS
LIN {X -0.358,Y -638.222,Z 828.637,A 0.000,B 0.000,C 90.000,E1 330.667} C_DIS
LIN {X -0.326,Y -643.421,Z 828.630,A 0.000,B 0.000,C 90.000,E1 329.410} C_DIS
LIN {X 0.200,Y -646.382,Z 828.626,A 0.000,B 0.000,C 90.000,E1 328.614} C_DIS
LIN {X -0.269,Y -649.856,Z 828.620,A 0.000,B 0.000,C 90.000,E1 327.661} C_DIS
LIN {X -0.229,Y -652.469,Z 828.616,A 0.000,B 0.000,C 90.000,E1 326.914} C_DIS
LIN {X -0.171,Y -656.401,Z 828.609,A 0.000,B 0.000,C 90.000,E1 325.674} C_DIS
LIN {X 0.305,Y -658.574,Z 828.605,A 0.000,B 0.000,C 90.000,E1 324.895} C_DIS
LIN {X 0.366,Y -661.200,Z 828.600,A 0.000,B 0.000,C 90.000,E1 323.909} C_DIS
LIN {X -0.073,Y -663.645,Z 828.594,A 0.000,B 0.000,C 90.000,E1 322.970} C_DIS
LIN {X 0.046,Y -665.887,Z 828.589,A 0.000,B 0.000,C 90.000,E1 321.984} C_DIS
LIN {X 0.092,Y -667.435,Z 828.585,A 0.000,B 0.000,C 90.000,E1 321.251} C_DIS
LIN {X -0.286,Y -670.238,Z 828.577,A 0.000,B 0.000,C 90.000,E1 319.828} C_DIS
LIN {X -0.182,Y -672.330,Z 828.570,A 0.000,B 0.000,C 90.000,E1 318.609} C_DIS
LIN {X -0.046,Y -674.312,Z 828.563,A 0.000,B 0.000,C 90.000,E1 317.391} C_DIS
LIN {X 0.028,Y -675.382,Z 828.559,A 0.000,B 0.000,C 90.000,E1 316.662} C_DIS
LIN {X -0.320,Y -676.669,Z 828.554,A 0.000,B 0.000,C 90.000,E1 315.729} C_DIS
LIN {X -0.181,Y -677.904,Z 828.549,A 0.000,B 0.000,C 90.000,E1 314.757} C_DIS
LIN {X 0.011,Y -679.264,Z 828.542,A 0.000,B 0.000,C 90.000,E1 313.542} C_DIS
LIN {X -0.249,Y -680.643,Z 828.535,A 0.000,B 0.000,C 90.000,E1 312.366} C_DIS
LIN {X 0.062,Y -682.207,Z 828.527,A 0.000,B 0.000,C 90.000,E1 310.906} C_DIS
LIN {X -0.086,Y -683.394,Z 828.521,A 0.000,B 0.000,C 90.000,E1 309.725} C_DIS
LIN {X -0.171,Y -684.680,Z 828.513,A 0.000,B 0.000,C 90.000,E1 308.302} C_DIS
LIN {X -0.088,Y -686.143,Z 828.503,A 0.000,B 0.000,C 90.000,E1 306.629} C_DIS
LIN {X 0.142,Y -687.287,Z 828.496,A 0.000,B 0.000,C 90.000,E1 305.185} C_DIS
LIN {X -0.153,Y -688.300,Z 828.488,A 0.000,B 0.000,C 90.000,E1 303.785} C_DIS
LIN {X -0.233,Y -689.493,Z 828.478,A 0.000,B 0.000,C 90.000,E1 302.133} C_DIS
LIN {X 0.160,Y -690.886,Z 828.468,A 0.000,B 0.000,C 90.000,E1 300.207} C_DIS
LIN {X 0.014,Y -692.094,Z 828.459,A 0.000,B 0.000,C 90.000,E1 298.565} C_DIS
LIN {X 0.128,Y -693.538,Z 828.448,A 0.000,B 0.000,C 90.000,E1 296.668} C_DIS
LIN {X -0.233,Y -694.731,Z 828.440,A 0.000,B 0.000,C 90.000,E1 295.283} C_DIS
LIN {X -0.147,Y -695.502,Z 828.435,A 0.000,B 0.000,C 90.000,E1 294.335} C_DIS
LIN {X 0.357,Y -695.582,Z 828.433,A 0.000,B 0.000,C 90.000,E1 293.823} C_DIS
LIN {X -0.308,Y -695.422,Z 828.431,A 0.000,B 0.000,C 90.000,E1 293.643} C_DIS
LIN {X 0.192,Y -694.574,Z 828.429,A 0.000,B 0.000,C 90.000,E1 293.131} C_DIS
LIN {X 0.167,Y -693.694,Z 828.427,A 0.000,B 0.000,C 90.000,E1 292.898} C_DIS
LIN {X -0.373,Y -691.380,Z 828.425,A 0.000,B 0.000,C 90.000,E1 292.589} C_DIS
LIN {X -0.137,Y -689.464,Z 828.424,A 0.000,B 0.000,C 90.000,E1 292.333} C_DIS
LIN {X -0.021,Y -688.038,Z 828.423,A 0.000,B 0.000,C 90.000,E1 292.206} C_DIS
LIN {X 0.073,Y -682.605,Z 828.422,A 0.000,B 0.000,C 90.000,E1 291.897} C_DIS
LIN {X -0.292,Y -680.881,Z 828.421,A 0.000,B 0.000,C 90.000,E1 291.844} C_DIS
LIN {X 0.301,Y -678.999,Z 828.421,A 0.000,B 0.000,C 90.000,E1 291.716} C_DIS
LIN {X -0.262,Y -670.847,Z 828.420,A 0.000,B 0.000,C 90.000,E1 291.535} C_DIS
LIN {X 0.087,Y -662.993,Z 828.419,A 0.000,B 0.000,C 90.000,E1 291.354} C_DIS
LIN {X -0.129,Y -653.703,Z 828.418,A 0.000,B 0.000,C 90.000,E1 291.227} C_DIS
LIN {X -0.176,Y -644.113,Z 828.417,A 0.000,B 0.000,C 90.000,E1 291.046} C_DIS
LIN {X 0.073,Y -634.189,Z 828.416,A 0.000,B 0.000,C 90.000,E1 290.791} C_DIS
LIN {X 0.049,Y -629.409,Z 828.415,A 0.000,B 0.000,C 90.000,E1 290.663} C_DIS
LIN {X 0.119,Y -622.492,Z 828.413,A 0.000,B 0.000,C 90.000,E1 290.375} C_DIS
LIN {X 0.133,Y -618.308,Z 828.412,A 0.000,B 0.000,C 90.000,E1 290.120} C_DIS
LIN {X 0.071,Y -618.209,Z 828.412,A 0.000,B 0.000,C 90.000,E1 290.120} C_DIS
LIN {X -0.210,Y -617.009,Z 828.411,A 0.000,B 0.000,C 90.000,E1 289.939} C_DIS
LIN {X -0.254,Y -617.009,Z 828.411,A 0.000,B 0.000,C 90.000,E1 289.939} C_DIS
LIN {X 0.156,Y -617.202,Z 828.410,A 0.000,B 0.000,C 90.000,E1 289.704} C_DIS
LIN {X 0.139,Y -617.453,Z 828.409,A 0.000,B 0.000,C 90.000,E1 289.577} C_DIS
LIN {X -0.138,Y -619.719,Z 828.406,A 0.000,B 0.000,C 90.000,E1 289.087} C_DIS
LIN {X -0.074,Y -624.742,Z 828.401,A 0.000,B 0.000,C 90.000,E1 288.236} C_DIS
LIN {X 0.086,Y -628.127,Z 828.398,A 0.000,B 0.000,C 90.000,E1 287.583} C_DIS
LIN {X -0.141,Y -631.000,Z 828.394,A 0.000,B 0.000,C 90.000,E1 286.968} C_DIS
LIN {X -0.112,Y -633.997,Z 828.390,A 0.000,B 0.000,C 90.000,E1 286.205} C_DIS
LIN {X 0.308,Y -635.728,Z 828.387,A 0.000,B 0.000,C 90.000,E1 285.662} C_DIS
LIN {X -0.219,Y -637.869,Z 828.383,A 0.000,B 0.000,C 90.000,E1 284.954} C_DIS
LIN {X 0.062,Y -639.041,Z 828.380,A 0.000,B 0.000,C 90.000,E1 284.426} C_DIS
LIN {X 0.346,Y -640.298,Z 828.376,A 0.000,B 0.000,C 90.000,E1 283.647} C_DIS
LIN {X 0.022,Y -640.900,Z 828.373,A 0.000,B 0.000,C 90.000,E1 283.175} C_DIS
LIN {X 0.325,Y -641.088,Z 828.370,A 0.000,B 0.000,C 90.000,E1 282.647} C_DIS
LIN {X 0.005,Y -640.963,Z 828.368,A 0.000,B 0.000,C 90.000,E1 282.175} C_DIS
LIN {X 0.180,Y -640.643,Z 828.365,A 0.000,B 0.000,C 90.000,E1 281.658} C_DIS
LIN {X 0.019,Y -640.451,Z 828.364,A 0.000,B 0.000,C 90.000,E1 281.422} C_DIS
LIN {X 0.321,Y -639.699,Z 828.361,A 0.000,B 0.000,C 90.000,E1 280.894} C_DIS
LIN {X -0.012,Y -638.676,Z 828.358,A 0.000,B 0.000,C 90.000,E1 280.423} C_DIS
LIN {X -0.295,Y -638.080,Z 828.357,A 0.000,B 0.000,C 90.000,E1 280.197} C_DIS
LIN {X -0.013,Y -636.592,Z 828.354,A 0.000,B 0.000,C 90.000,E1 279.670} C_DIS
LIN {X 0.152,Y -634.699,Z 828.351,A 0.000,B 0.000,C 90.000,E1 279.151} C_DIS
LIN {X 0.261,Y -631.739,Z 828.347,A 0.000,B 0.000,C 90.000,E1 278.511} C_DIS
LIN {X -0.227,Y -628.917,Z 828.345,A 0.000,B 0.000,C 90.000,E1 278.049} C_DIS
LIN {X -0.176,Y -624.559,Z 828.341,A 0.000,B 0.000,C 90.000,E1 277.409} C_DIS
LIN {X 0.064,Y -621.542,Z 828.339,A 0.000,B 0.000,C 90.000,E1 277.004} C_DIS
LIN {X -0.245,Y -619.104,Z 828.338,A 0.000,B 0.000,C 90.000,E1 276.777} C_DIS
LIN {X 0.075,Y -615.325,Z 828.336,A 0.000,B 0.000,C 90.000,E1 276.372} C_DIS
LIN {X -0.040,Y -613.889,Z 828.335,A 0.000,B 0.000,C 90.000,E1 276.258} C_DIS
LIN {X 0.181,Y -607.807,Z 828.332,A 0.000,B 0.000,C 90.000,E1 275.796} C_DIS
LIN {X 0.272,Y -606.098,Z 828.332,A 0.000,B 0.000,C 90.000,E1 275.682} C_DIS
LIN {X -0.137,Y -597.563,Z 828.329,A 0.000,B 0.000,C 90.000,E1 275.277} C_DIS
LIN {X -0.240,Y -592.251,Z 828.328,A 0.000,B 0.000,C 90.000,E1 275.049} C_DIS
LIN {X -0.207,Y -585.316,Z 828.326,A 0.000,B 0.000,C 90.000,E1 274.759} C_DIS
LIN {X 0.121,Y -579.623,Z 828.325,A 0.000,B 0.000,C 90.000,E1 274.531} C_DIS
LIN {X -0.249,Y -573.491,Z 828.324,A 0.000,B 0.000,C 90.000,E1 274.416} C_DIS
LIN {X -0.108,Y -571.097,Z 828.324,A 0.000,B 0.000,C 90.000,E1 274.359} C_DIS
LIN {X -0.211,Y -565.671,Z 828.324,A 0.000,B 0.000,C 90.000,E1 274.302} C_DIS
LIN {X 0.200,Y -559.347,Z 828.324,A 0.000,B 0.000,C 90.000,E1 274.245} C_DIS
LIN {X 0.168,Y -553.430,Z 828.324,A 0.000,B 0.000,C 90.000,E1 274.245} C_DIS
LIN {X 0.135,Y -550.287,Z 828.323,A 0.000,B 0.000,C 90.000,E1 274.188} C_DIS
LIN {X 0.100,Y -550.261,Z 828.323,A 0.000,B 0.000,C 90.000,E1 274.188} C_DIS
LIN {X -0.005,Y -549.660,Z 828.322,A 0.000,B 0.000,C 90.000,E1 274.012} C_DIS
LIN {X 0.062,Y -548.431,Z 828.317,A 0.000,B 0.000,C 90.000,E1 272.980} C_DIS
LIN {X -0.054,Y -546.385,Z 828.303,A 0.000,B 0.000,C 90.000,E1 270.458} C_DIS
LIN {X 0.193,Y -545.150,Z 828.293,A 0.000,B 0.000,C 90.000,E1 268.740} C_DIS
LIN {X -0.187,Y -544.354,Z 828.287,A 0.000,B 0.000,C 90.000,E1 267.650} C_DIS
LIN {X 0.061,Y -543.271,Z 828.277,A 0.000,B 0.000,C 90.000,E1 265.927} C_DIS
LIN {X 0.263,Y -542.335,Z 828.270,A 0.000,B 0.000,C 90.000,E1 264.489} C_DIS
LIN {X -0.108,Y -541.552,Z 828.263,A 0.000,B 0.000,C 90.000,E1 263.394} C_DIS
LIN {X -0.027,Y -540.826,Z 828.259,A 0.000,B 0.000,C 90.000,E1 262.534} C_DIS
LIN {X -0.145,Y -538.962,Z 828.247,A 0.000,B 0.000,C 90.000,E1 260.557} C_DIS
LIN {X 0.165,Y -537.297,Z 828.238,A 0.000,B 0.000,C 90.000,E1 258.814} C_DIS
LIN {X 0.113,Y -535.012,Z 828.225,A 0.000,B 0.000,C 90.000,E1 256.533} C_DIS
LIN {X 0.189,Y -532.740,Z 828.214,A 0.000,B 0.000,C 90.000,E1 254.519} C_DIS
LIN {X 0.146,Y -531.128,Z 828.206,A 0.000,B 0.000,C 90.000,E1 253.087} C_DIS
LIN {X -0.258,Y -528.982,Z 828.197,A 0.000,B 0.000,C 90.000,E1 251.402} C_DIS
LIN {X -0.034,Y -527.107,Z 828.189,A 0.000,B 0.000,C 90.000,E1 249.934} C_DIS
LIN {X 0.159,Y -525.064,Z 828.180,A 0.000,B 0.000,C 90.000,E1 248.465} C_DIS
LIN {X -0.021,Y -522.591,Z 828.171,A 0.000,B 0.000,C 90.000,E1 246.741} C_DIS
LIN {X 0.009,Y -520.298,Z 828.163,A 0.000,B 0.000,C 90.000,E1 245.281} C_DIS
LIN {X 0.007,Y -517.976,Z 828.155,A 0.000,B 0.000,C 90.000,E1 243.819} C_DIS
LIN {X -0.167,Y -515.921,Z 828.148,A 0.000,B 0.000,C 90.000,E1 242.666} C_DIS
LIN {X -0.022,Y -513.314,Z 828.140,A 0.000,B 0.000,C 90.000,E1 241.179} C_DIS
LIN {X 0.315,Y -510.618,Z 828.132,A 0.000,B 0.000,C 90.000,E1 239.665} C_DIS
LIN {X -0.173,Y -508.434,Z 828.125,A 0.000,B 0.000,C 90.000,E1 238.535} C_DIS
LIN {X 0.003,Y -506.078,Z 828.119,A 0.000,B 0.000,C 90.000,E1 237.327} C_DIS
LIN {X 0.302,Y -502.903,Z 828.110,A 0.000,B 0.000,C 90.000,E1 235.801} C_DIS
LIN {X -0.327,Y -500.892,Z 828.105,A 0.000,B 0.000,C 90.000,E1 234.975} C_DIS
LIN {X 0.161,Y -497.433,Z 828.097,A 0.000,B 0.000,C 90.000,E1 233.417} C_DIS
LIN {X 0.040,Y -493.118,Z 828.087,A 0.000,B 0.000,C 90.000,E1 231.618} C_DIS
LIN {X -0.253,Y -488.748,Z 828.077,A 0.000,B 0.000,C 90.000,E1 229.828} C_DIS
LIN {X 0.222,Y -485.236,Z 828.068,A 0.000,B 0.000,C 90.000,E1 228.243} C_DIS
LIN {X -0.092,Y -481.760,Z 828.060,A 0.000,B 0.000,C 90.000,E1 226.743} C_DIS
LIN {X -0.114,Y -476.383,Z 828.046,A 0.000,B 0.000,C 90.000,E1 224.271} C_DIS
LIN {X 0.042,Y -471.024,Z 828.032,A 0.000,B 0.000,C 90.000,E1 221.757} C_DIS
LIN {X -0.002,Y -466.334,Z 828.020,A 0.000,B 0.000,C 90.000,E1 219.564} C_DIS
LIN {X 0.103,Y -463.077,Z 828.011,A 0.000,B 0.000,C 90.000,E1 217.971} C_DIS
LIN {X -0.110,Y -459.128,Z 828.000,A 0.000,B 0.000,C 90.000,E1 216.091} C_DIS
LIN {X -0.042,Y -455.822,Z 827.992,A 0.000,B 0.000,C 90.000,E1 214.485} C_DIS
LIN {X 0.139,Y -451.014,Z 827.979,A 0.000,B 0.000,C 90.000,E1 212.212} C_DIS
LIN {X 0.172,Y -447.671,Z 827.970,A 0.000,B 0.000,C 90.000,E1 210.590} C_DIS
LIN {X -0.188,Y -443.119,Z 827.957,A 0.000,B 0.000,C 90.000,E1 208.359} C_DIS
LIN {X 0.034,Y -439.926,Z 827.948,A 0.000,B 0.000,C 90.000,E1 206.693} C_DIS
LIN {X 0.192,Y -436.617,Z 827.939,A 0.000,B 0.000,C 90.000,E1 205.027} C_DIS
LIN {X -0.084,Y -432.540,Z 827.928,A 0.000,B 0.000,C 90.000,E1 203.078} C_DIS
LIN {X 0.175,Y -428.703,Z 827.917,A 0.000,B 0.000,C 90.000,E1 201.046} C_DIS
LIN {X -0.004,Y -425.475,Z 827.908,A 0.000,B 0.000,C 90.000,E1 199.396} C_DIS
LIN {X 0.145,Y -422.140,Z 827.898,A 0.000,B 0.000,C 90.000,E1 197.692} C_DIS
LIN {X -0.080,Y -419.578,Z 827.891,A 0.000,B 0.000,C 90.000,E1 196.370} C_DIS
LIN {X -0.217,Y -415.074,Z 827.878,A 0.000,B 0.000,C 90.000,E1 194.008} C_DIS
LIN {X -0.193,Y -411.040,Z 827.866,A 0.000,B 0.000,C 90.000,E1 191.951} C_DIS
LIN {X 0.050,Y -407.098,Z 827.855,A 0.000,B 0.000,C 90.000,E1 189.849} C_DIS
LIN {X 0.114,Y -403.847,Z 827.845,A 0.000,B 0.000,C 90.000,E1 188.106} C_DIS
LIN {X -0.003,Y -399.949,Z 827.834,A 0.000,B 0.000,C 90.000,E1 186.030} C_DIS
LIN {X 0.199,Y -392.988,Z 827.810,A 0.000,B 0.000,C 90.000,E1 181.776} C_DIS
LIN {X -0.130,Y -388.809,Z 827.792,A 0.000,B 0.000,C 90.000,E1 178.625} C_DIS
LIN {X -0.177,Y -386.581,Z 827.782,A 0.000,B 0.000,C 90.000,E1 176.846} C_DIS
LIN {X 0.006,Y -383.991,Z 827.770,A 0.000,B 0.000,C 90.000,E1 174.666} C_DIS
LIN {X -0.174,Y -379.991,Z 827.750,A 0.000,B 0.000,C 90.000,E1 171.084} C_DIS
LIN {X -0.026,Y -377.619,Z 827.736,A 0.000,B 0.000,C 90.000,E1 168.522} C_DIS
LIN {X 0.087,Y -375.103,Z 827.720,A 0.000,B 0.000,C 90.000,E1 165.589} C_DIS
LIN {X -0.019,Y -372.702,Z 827.692,A 0.000,B 0.000,C 90.000,E1 160.477} C_DIS
LIN {X -0.042,Y -372.854,Z 827.681,A 0.000,B 0.000,C 90.000,E1 158.646} C_DIS
LIN {X 0.074,Y -373.755,Z 827.671,A 0.000,B 0.000,C 90.000,E1 156.794} C_DIS
LIN {X -0.073,Y -374.805,Z 827.665,A 0.000,B 0.000,C 90.000,E1 155.717} C_DIS
LIN {X 0.012,Y -375.762,Z 827.661,A 0.000,B 0.000,C 90.000,E1 154.973} C_DIS
LIN {X 0.100,Y -377.012,Z 827.657,A 0.000,B 0.000,C 90.000,E1 154.229} C_DIS
LIN {X 0.022,Y -378.555,Z 827.653,A 0.000,B 0.000,C 90.000,E1 153.512} C_DIS
